// TwinCAT 3 PLC project MTCS
// ProgramVersion: 3.1.4020.1
// libraries:
//   Tc2_ControllerToolbox, * (Beckhoff Automation GmbH)
//   Tc2_Drive, * (Beckhoff Automation GmbH)
//   Tc2_EtherCAT, * (Beckhoff Automation GmbH)
//   Tc2_Math, * (Beckhoff Automation GmbH)
//   Tc2_MC2, * (Beckhoff Automation GmbH)
//   Tc2_MC2_Drive, * (Beckhoff Automation GmbH)
//   Tc2_SerialCom, * (Beckhoff Automation GmbH)
//   Tc2_Standard, * (Beckhoff Automation GmbH)
//   Tc2_System, * (Beckhoff Automation GmbH)
//   Tc2_Utilities, * (Beckhoff Automation GmbH)
//   Tc2_XmlDataSrv, * (Beckhoff Automation GmbH)
//   Tc3_Interfaces, * (Beckhoff Automation GmbH)
//   Tc3_Module, * (Beckhoff Automation GmbH)
//   VisuDialogs, * (System)
//   VisuUserMgmt, * (System)
// project tree:
//   / GlobalTextList.TcGTLO, PlcFastTask.TcTTO, PlcTask.TcTTO, Visualization Manager.TcVMO (not stored), VISU_TASK.TcTTO
//   GVLs/ GLOBAL.TcGVL, REMANENT.TcGVL
//   MTCS/Axes/Generated/mtcs_axes/Configs/ AxesAzimuthConfig.TcDUT (not stored), AxesConfig.TcDUT (not stored), AxesElevationConfig.TcDUT (not stored), AxesKnownPositionConfig.TcDUT (not stored), AxesKnownPositionsConfig.TcDUT (not stored), AxesLocalConditionsConfig.TcDUT (not stored), AxesLocationConfig.TcDUT (not stored), AxesPointingModelConfig.TcDUT (not stored), AxesRotationConfig.TcDUT (not stored)
//   MTCS/Axes/Generated/mtcs_axes/Enums/ AxesAlphaUnits.TcDUT (not stored), AxesDeltaUnits.TcDUT (not stored), AxesIds.TcDUT (not stored), AxesMoveUnits.TcDUT (not stored), AxesMoveVelocityUnits.TcDUT (not stored), AxesMuUnits.TcDUT (not stored), AxesRotatorActivity.TcDUT (not stored)
//   MTCS/Axes/Generated/mtcs_axes/Processes/Args/ AxesEnablePointingModelProcessArgs.TcDUT (not stored), AxesMoveAbsoluteProcessArgs.TcDUT (not stored), AxesMoveKnownPositionProcessArgs.TcDUT (not stored), AxesMoveOutOfLimitSwitchProcessArgs.TcDUT (not stored), AxesMoveRelativeProcessArgs.TcDUT (not stored), AxesMoveVelocityProcessArgs.TcDUT (not stored), AxesMultiMoveProcessArgs.TcDUT (not stored), AxesPointProcessArgs.TcDUT (not stored), AxesPointRelativeProcessArgs.TcDUT (not stored), AxesMultiPowerOnProcessArgs.TcDUT (not stored), AxesSetAlphaDeltaVelocityProcessArgs.TcDUT (not stored), AxesSetPositionProcessArgs.TcDUT (not stored), AxesSetTargetProcessArgs.TcDUT (not stored), AxesUnlockBrakeProcessArgs.TcDUT (not stored)
//   MTCS/Axes/Generated/mtcs_axes/Processes/ AxesDoHomingProcess.TcPOU (not stored), AxesEnablePointingModelProcess.TcPOU (not stored), AxesMoveAbsoluteProcess.TcPOU (not stored), AxesMoveKnownPositionProcess.TcPOU (not stored), AxesMoveOutOfLimitSwitchProcess.TcPOU (not stored), AxesMoveRelativeProcess.TcPOU (not stored), AxesMoveVelocityProcess.TcPOU (not stored), AxesMultiMoveProcess.TcPOU (not stored), AxesPointProcess.TcPOU (not stored), AxesPointRelativeProcess.TcPOU (not stored), AxesPowerOffProcess.TcPOU (not stored), AxesPowerOnProcess.TcPOU (not stored), AxesMultiPowerOnProcess.TcPOU (not stored), AxesSetAlphaDeltaVelocityProcess.TcPOU (not stored), AxesSetPositionProcess.TcPOU (not stored), AxesSetTargetProcess.TcPOU (not stored), AxesStopProcess.TcPOU (not stored), AxesUnlockBrakeProcess.TcPOU (not stored)
//   MTCS/Axes/Generated/mtcs_axes/StateMachines/Parts/ AxesAzimuthAxisParts.TcDUT (not stored), AxesElevationAxisParts.TcDUT (not stored), AxesIOParts.TcDUT (not stored), AxesParts.TcDUT (not stored), AxesPointingModelSetupParts.TcDUT (not stored), AxesPointingModelsSetupParts.TcDUT (not stored), AxesRotationAxisParts.TcDUT (not stored)
//   MTCS/Axes/Generated/mtcs_axes/StateMachines/Processes/ AxesAzimuthAxisProcesses.TcDUT (not stored), AxesElevationAxisProcesses.TcDUT (not stored), AxesProcesses.TcDUT (not stored), AxesRotationAxisProcesses.TcDUT (not stored)
//   MTCS/Axes/Generated/mtcs_axes/StateMachines/ SM_Axes.TcPOU (not stored), SM_AxesAzimuthAxis.TcPOU (not stored), SM_AxesElevationAxis.TcPOU (not stored), SM_AxesFeedback.TcPOU (not stored), SM_AxesIO.TcPOU (not stored), SM_AxesPointingModelSetup.TcPOU (not stored), SM_AxesPointingModelsSetup.TcPOU (not stored), SM_AxesRotationAxis.TcPOU (not stored), SM_AxesTarget.TcPOU (not stored)
//   MTCS/Axes/Generated/mtcs_axes/StateMachines/Statuses/ AxesAzimuthAxisStatuses.TcDUT (not stored), AxesElevationAxisStatuses.TcDUT (not stored), AxesFeedbackStatuses.TcDUT (not stored), AxesIOStatuses.TcDUT (not stored), AxesPointingModelsSetupStatuses.TcDUT (not stored), AxesRotationAxisStatuses.TcDUT (not stored), AxesStatuses.TcDUT (not stored), AxesTargetStatuses.TcDUT (not stored)
//   MTCS/Axes/Helper/ ARCSEC_TO_RAD.TcPOU, AxesDeltaUnitsToDeg.TcPOU, AxesGetKnownPositionConfig.TcPOU, AxesLidaPositionToValue.TcPOU, AxesMoveRelativeCalculator.TcPOU, AxesMoveVelocityUnitsToString.TcPOU, AxesMoveAbsoluteCalculator.TcPOU, AxesSlalibSmoothener.TcPOU, AxesQuickStopHelper.TcPOU, AxesUnlockBrakeHelper.TcPOU, HOUR_TO_DEG.TcPOU, AxesAlphaUnitsToDeg.TcPOU, AxesMoveVelocityUnitsToDegPerSec.TcPOU, HMS_TO_DEG.TcPOU, DEG_TO_ARCSEC.TcPOU, DMS_TO_DEG.TcPOU, MILLIARCSEC_TO_DEG.TcPOU, ARCSEC_TO_DEG.TcPOU, AverageAndRmsCalculator.TcPOU, AxesCalculateLidaAveragePosition.TcPOU, AxesLidaValueToPosition.TcPOU, AxesMuUnitsToDegPerYear.TcPOU, AxesSSIValueToPosition.TcPOU, AxesExternalSetpointGenerator.TcPOU, AxesFastTaskAxisIO.TcDUT, AxesMoveOutOfLimitSwitchHelper.TcPOU, AxesPowerOffHelper.TcPOU, AxesHomingHelper.TcPOU, AxesPowerOnHelper.TcPOU, AxesStopHelper.TcPOU, AxesSetPositionHelper.TcPOU, AxesTorqueSetpointGenerator.TcPOU, AxesCalculateTorqueCommandValue.TcPOU, AxesTPointCalculations.TcPOU, HoursMinutesSeconds.TcDUT, DegreesMinutesSeconds.TcDUT, AxesMoveUnitsToDeg.TcPOU, RAD_TO_DEG.TcPOU, DEG_TO_RAD_REAL.TcPOU, CELSIUS_TO_KELVIN.TcPOU, DEG_TO_RAD.TcPOU, RAD_TO_HOUR.TcPOU, TmcAxesErrorsToString.TcPOU
//   MTCS/Axes/StateMachines/ Axes.TcPOU, AxesElevationAxis.TcPOU, AxesRotationAxis.TcPOU, AxesIO.TcPOU, AxesPointingModelsSetup.TcPOU, AxesAzimuthAxis.TcPOU, AxesPointingModelSetup.TcPOU, AxesTarget.TcPOU, AxesFeedback.TcPOU
//   MTCS/Axes/Visu/Tube/ VISU_Tube_Rotator.TcVIS (not stored), VISU_Tube_Side.TcVIS (not stored), VISU_Tube_Top_0.TcVIS (not stored), VISU_Tube_Top_fork.TcVIS (not stored), VISU_Tube_Top_1.TcVIS (not stored), VISU_Tube_Top_9.TcVIS (not stored), VISU_Tube_Top_10.TcVIS (not stored), VISU_Tube_Top_11.TcVIS (not stored), VISU_Tube_Top_12.TcVIS (not stored), VISU_Tube_Top_14.TcVIS (not stored), VISU_Tube_Top_2.TcVIS (not stored), VISU_Tube_Top_3.TcVIS (not stored), VISU_Tube_Top_13.TcVIS (not stored), VISU_Tube_Top_4.TcVIS (not stored), VISU_Tube_Top_5.TcVIS (not stored), VISU_Tube_Top_6.TcVIS (not stored), VISU_Tube_Top_7.TcVIS (not stored), VISU_Tube_Top_8.TcVIS (not stored), VISU_Tube_Top.TcVIS (not stored)
//   MTCS/Axes/Visu/ VISU_AxesAzimuthAxis.TcVIS, VISU_AxesAzimuthAxis_AbsoluteEncoder.TcVIS, VISU_AxesAzimuthAxis_Processes.TcVIS, VISU_AxesConfig_KnownPosition.TcVIS, VISU_AxesConfig_KnownPositions.TcVIS, VISU_AxesImage.TcVIS, VISU_AxesManual_Offsets_AlphaDeltaRot.TcVIS, VISU_AxesManual_Offsets_OLD.TcVIS, VISU_AxesRotationAxis_Processes.TcVIS, VISU_AxesRotationAxis_Overview.TcVIS, VISU_AxesElevationAxis_Processes.TcVIS, VISU_AxesManual_MoveVelocity.TcVIS, VISU_AxesManual_Offsets_AziEleRot.TcVIS, VISU_AxesManual_Joystick_AziEle.TcVIS, VISU_AxesManual_Joystick_Rot.TcVIS, VISU_AxesManual_Positions.TcVIS, VISU_AxesManual_MoveAbsolute.TcVIS, VISU_Axes_Commands_Power.TcVIS, VISU_AxesElevationAxis_Overview.TcVIS, VISU_AxesElevationAxis_AbsoluteEncoder.TcVIS, VISU_AxesElevationAxis_Lidas.TcVIS, VISU_AxesAzimuthAxis_Overview.TcVIS, VISU_AxesAzimuthAxis_Lidas.TcVIS, VISU_AxesConfig_Azimuth_1.TcVIS, VISU_AxesConfig_Azimuth_3.TcVIS, VISU_AxesConfig_Rotation_2.TcVIS, VISU_AxesConfig_Rotation_1.TcVIS, VISU_AxesConfig_Elevation_2.TcVIS, VISU_AxesConfig_Elevation_1.TcVIS, VISU_AxesConfig_Azimuth_2.TcVIS, VISU_AxesConfig_FilterWheel.TcVIS, VISU_AxesElevationAxis.TcVIS, VISU_AxesExternalSetpointGenerator.TcVIS, VISU_AxesRotationAxis.TcVIS, VISU_AxesManual.TcVIS, VISU_AxesConfig.TcVIS, VISU_AxesAxes.TcVIS, VISU_AxesAdvanced.TcVIS, VISU_AxesPointingModelConfig_part1.TcVIS, VISU_AxesPointingModelConfig_part2.TcVIS, VISU_AxesPointingModelSetup.TcVIS, VISU_AxesConfig_General.TcVIS, VISU_AxesConfig_Location.TcVIS, VISU_AxesConfig_LocalConditions.TcVIS, VISU_AxesFromCpp_Target.TcVIS, VISU_AxesIO.TcVIS, VISU_Axes.TcVIS, VISU_AxesOverview.TcVIS, VISU_AxesMultiMoveProcess.TcVIS, VISU_AxesPointingModelsSetup.TcVIS, VISU_AxesPointDialog.TcVIS, VISU_AxesTarget.TcVIS, VISU_AxesSetTargetDialog.TcVIS, VISU_AxesFromCpp.TcVIS, VISU_Axes_Commands_Reset.TcVIS, VISU_Axes_Commands_Brake.TcVIS, VISU_Axes_Commands_Movement.TcVIS, VISU_Axes_Commands_DoHoming.TcVIS, VISU_Axes_stats.TcVIS
//   MTCS/Axes/Widgets/ AxesAlphaWidget.TcPOU, AxesAngleWidget.TcPOU, AxesDialogRotUnits.TcDUT, AxesDialogRotUnitsTextList.TcTLO, AxesMoveAlphaDeltaProcessUnitsTextList.TcTLO, AxesPointRelativeProcessWidget.TcPOU, AxesRotationAxisTabs.TcDUT, AxesManualTabs.TcDUT, AxesElevationAxisTabs.TcDUT, AxesDeltaWidget.TcPOU, AxesAzimuthAxisTabs.TcDUT, AxesDialogAlphaUnitsTextList.TcTLO, AxesDialogSignTextList.TcTLO, AxesManualJoystickAziEleWidget.TcPOU, AxesManualJoystickRotWidget.TcPOU, AxesManualOffsetsWidget.TcPOU, AxesManualMoveVelocityWidget.TcPOU, AxesManualPositionsWidget.TcPOU, AxesManualMoveAbsoluteWidget.TcPOU, AxesMoveUnitsTextList.TcTLO, AxesMoveVelocityUnitsTextList.TcTLO, AxesMuUnitsTextList.TcTLO, AxesDialogDeltaUnitsTextList.TcTLO, AxesDialogSign.TcDUT, AxesElevationAxisWidget.TcPOU, AxesConfigTextList.TcTLO, AxesAxesTabs.TcDUT, AxesAxesWidget.TcPOU, AxesImageWidget.TcPOU, AxesManualWidget.TcPOU, AxesMultiMoveProcessWidget.TcPOU, AxesRotationAxisWidget.TcPOU, AxesPointingModelSetupPartsTextList.TcTLO, AxesIOWidget.TcPOU, AxesPointingModelSetupWidget.TcPOU, AxesMoveProcessUnitsTextList.TcTLO, AxesMoveProcessWidgetUnits.TcDUT, AxesPointingModelsSetupWidget.TcPOU, AxesAzimuthAxisWidget.TcPOU, AxesDialogAlphaUnits.TcDUT, AxesDialogDeltaUnits.TcDUT, AxesSetTargetDialogWidget.TcPOU, AxesPointDialogWidget.TcPOU, AxesTabs.TcDUT, AxesTargetWidget.TcPOU, AxesFeedbackWidget.TcPOU, AxesWidget.TcPOU
//   MTCS/Common/Generated/mtcs_common/Configs/ FaulhaberDriveConfig.TcDUT (not stored), HiHiLoLoAlarmConfig.TcDUT (not stored), InstrumentConfig.TcDUT (not stored), MeasurementConfig.TcDUT (not stored)
//   MTCS/Common/Generated/mtcs_common/Enums/ DriveBrakeStates.TcDUT (not stored), DriveOperatingModes.TcDUT (not stored), InitializationStates.TcDUT (not stored), LimitSwitches.TcDUT (not stored), OperatingStates.TcDUT (not stored), OperatorStates.TcDUT (not stored), RequestResults.TcDUT (not stored), Units.TcDUT (not stored)
//   MTCS/Common/Generated/mtcs_common/Processes/ ActivateProcess.TcPOU (not stored), ChangeOperatingStateProcess.TcPOU (not stored), ChangeOperatorStateProcess.TcPOU (not stored), ChangeSetpointProcess.TcPOU (not stored), McMoveAbsoluteProcess.TcPOU (not stored), McMoveRelativeProcess.TcPOU (not stored), McMoveVelocityProcess.TcPOU (not stored), McPowerProcess.TcPOU (not stored), McProcess.TcPOU (not stored), McReadBoolParameter.TcPOU (not stored), McReadParameter.TcPOU (not stored), McSetPositionProcess.TcPOU (not stored), McStopProcess.TcPOU (not stored), McWriteBoolParameter.TcPOU (not stored), McWriteParameter.TcPOU (not stored), Process.TcPOU (not stored), ReadXmlProcess.TcPOU (not stored), SDOReadProcess.TcPOU (not stored), SDOWriteProcess.TcPOU (not stored), SetBrakeProcess.TcPOU (not stored), SetEnabledProcess.TcPOU (not stored), SoEReadProcess.TcPOU (not stored), SoEResetProcess.TcPOU (not stored), SoEWriteProcess.TcPOU (not stored), WriteXmlProcess.TcPOU (not stored)
//   MTCS/Common/Generated/mtcs_common/Processes/Args/ ChangeOperatingStateProcessArgs.TcDUT (not stored), ChangeOperatorStateProcessArgs.TcDUT (not stored), ChangeSetpointProcessArgs.TcDUT (not stored), McMoveAbsoluteProcessArgs.TcDUT (not stored), McMoveRelativeProcessArgs.TcDUT (not stored), McMoveVelocityProcessArgs.TcDUT (not stored), McPowerProcessArgs.TcDUT (not stored), McReadBoolParameterArgs.TcDUT (not stored), McReadParameterArgs.TcDUT (not stored), McSetPositionProcessArgs.TcDUT (not stored), McStopProcessArgs.TcDUT (not stored), McWriteBoolParameterArgs.TcDUT (not stored), McWriteParameterArgs.TcDUT (not stored), ReadXmlProcessArgs.TcDUT (not stored), SDOReadProcessArgs.TcDUT (not stored), SDOWriteProcessArgs.TcDUT (not stored), SetBrakeProcessArgs.TcDUT (not stored), SetEnabledProcessArgs.TcDUT (not stored), SoEReadProcessArgs.TcDUT (not stored), SoEWriteProcessArgs.TcDUT (not stored), WriteXmlProcessArgs.TcDUT (not stored)
//   MTCS/Common/Generated/mtcs_common/StateMachines/Parts/ AX52XXDriveParts.TcDUT (not stored)
//   MTCS/Common/Generated/mtcs_common/StateMachines/Processes/ AX52XXDriveChannelProcesses.TcDUT (not stored), BaseAxisProcesses.TcDUT (not stored), ConfigManagerProcesses.TcDUT (not stored), FaulhaberDriveProcesses.TcDUT (not stored), IncrementalEncoderProcesses.TcDUT (not stored), SimpleRelayProcesses.TcDUT (not stored)
//   MTCS/Common/Generated/mtcs_common/StateMachines/ SM_AngularAcceleration.TcPOU (not stored), SM_AngularAxis.TcPOU (not stored), SM_AngularPosition.TcPOU (not stored), SM_AngularVelocity.TcPOU (not stored), SM_AverageCurrent.TcPOU (not stored), SM_AX52XXDrive.TcPOU (not stored), SM_AX52XXDriveChannel.TcPOU (not stored), SM_BaseAxis.TcPOU (not stored), SM_BaseMcProcess.TcPOU (not stored), SM_BaseProcess.TcPOU (not stored), SM_BaseXmlDataSrvProcess.TcPOU (not stored), SM_CANopenBus.TcPOU (not stored), SM_ConfigManager.TcPOU (not stored), SM_Current.TcPOU (not stored), SM_CurrentMeasurement.TcPOU (not stored), SM_EtherCatDevice.TcPOU (not stored), SM_FaulhaberDrive.TcPOU (not stored), SM_Force.TcPOU (not stored), SM_ForceMeasurement.TcPOU (not stored), SM_Fraction.TcPOU (not stored), SM_Frequency.TcPOU (not stored), SM_FrequencyMeasurement.TcPOU (not stored), SM_GForce.TcPOU (not stored), SM_GForceMeasurement.TcPOU (not stored), SM_IncrementalEncoder.TcPOU (not stored), SM_LinearAxis.TcPOU (not stored), SM_LinearPosition.TcPOU (not stored), SM_LinearPositionMeasurement16.TcPOU (not stored), SM_LinearPositionMeasurementU32.TcPOU (not stored), SM_LinearVelocity.TcPOU (not stored), SM_Pressure.TcPOU (not stored), SM_PressureMeasurement.TcPOU (not stored), SM_ProcessStep.TcPOU (not stored), SM_QuantityValue.TcPOU (not stored), SM_RelativeHumidityMeasurement.TcPOU (not stored), SM_SimpleRelay.TcPOU (not stored), SM_SSIEncoder.TcPOU (not stored), SM_Temperature.TcPOU (not stored), SM_TemperatureMeasurement.TcPOU (not stored), SM_Torque.TcPOU (not stored), SM_TorqueLimit.TcPOU (not stored), SM_Voltage.TcPOU (not stored), SM_VoltageMeasurement.TcPOU (not stored)
//   MTCS/Common/Generated/mtcs_common/StateMachines/Statuses/ AX52XXDriveChannelStatuses.TcDUT (not stored), AX52XXDriveStatuses.TcDUT (not stored), BaseAxisStatuses.TcDUT (not stored), BaseProcessStatuses.TcDUT (not stored), CANopenBusStatuses.TcDUT (not stored), ConfigManagerStatuses.TcDUT (not stored), CurrentMeasurementStatuses.TcDUT (not stored), EtherCatDeviceStatuses.TcDUT (not stored), FaulhaberDriveStatuses.TcDUT (not stored), ForceMeasurementStatuses.TcDUT (not stored), FrequencyMeasurementStatuses.TcDUT (not stored), GForceMeasurementStatuses.TcDUT (not stored), IncrementalEncoderStatuses.TcDUT (not stored), LinearPositionMeasurement16Statuses.TcDUT (not stored), LinearPositionMeasurementU32Statuses.TcDUT (not stored), PressureMeasurementStatuses.TcDUT (not stored), ProcessStepStatuses.TcDUT (not stored), RelativeHumidityMeasurementStatuses.TcDUT (not stored), SimpleRelayStatuses.TcDUT (not stored), SSIEncoderStatuses.TcDUT (not stored), TemperatureMeasurementStatuses.TcDUT (not stored), VoltageMeasurementStatuses.TcDUT (not stored)
//   MTCS/Common/Generated/mtcs_common/Statuses/ ActivityStatus.TcPOU (not stored), ApertureStatus.TcPOU (not stored), BusyStatus.TcPOU (not stored), EnabledStatus.TcPOU (not stored), HealthStatus.TcPOU (not stored), HiHiLoLoAlarmStatus.TcPOU (not stored), InitializationStatus.TcPOU (not stored), MotionStatus.TcPOU (not stored), OpeningStatus.TcPOU (not stored), OperatingStatus.TcPOU (not stored), OperatorStatus.TcPOU (not stored), PoweredStatus.TcPOU (not stored), StartedStatus.TcPOU (not stored)
//   MTCS/Common/HelperCode/ BusyToColor.TcPOU, ComErrorToString.TcPOU, DegToRad.TcPOU, DriveBrakeStatesToString.TcPOU, DriveOperatingModesToString.TcPOU, HealthBusyToColor.TcPOU, HealthToColor.TcPOU, InitializationStatusToString.TcPOU, MeasurementToString.TcPOU, MeasurementToStatus.TcPOU, RadToDeg.TcPOU, SerialLine.TcPOU, StatusColor.TcDUT, SystemToColor.TcPOU
//   MTCS/Common/StateMachines/ AngularAxis.TcPOU, AngularPosition.TcPOU, AngularVelocity.TcPOU, AngularAcceleration.TcPOU, AverageCurrent.TcPOU, AX52XXDrive.TcPOU, AX52XXDriveChannel.TcPOU, BaseAxis.TcPOU, BaseMcProcess.TcPOU, BaseProcess.TcPOU, BaseXmlDataSrvProcess.TcPOU, CANopenBus.TcPOU, ConfigManager.TcPOU, Current.TcPOU, CurrentMeasurement.TcPOU, Torque.TcPOU, GForce.TcPOU, LinearPositionMeasurement16.TcPOU, EtherCatDevice.TcPOU, FaulhaberDrive.TcPOU, Force.TcPOU, ForceMeasurement.TcPOU, Frequency.TcPOU, FrequencyMeasurement.TcPOU, Fraction.TcPOU, IncrementalEncoder.TcPOU, LinearAxis.TcPOU, LinearPosition.TcPOU, LinearPositionMeasurementU32.TcPOU, LinearVelocity.TcPOU, Pressure.TcPOU, PressureMeasurement.TcPOU, ProcessStep.TcPOU, QuantityValue.TcPOU, RelativeHumidityMeasurement.TcPOU, SimpleRelay.TcPOU, SSIEncoder.TcPOU, Temperature.TcPOU, TemperatureMeasurement.TcPOU, TorqueLimit.TcPOU, Voltage.TcPOU, VoltageMeasurement.TcPOU, GForceMeasurement.TcPOU
//   MTCS/Common/Visu/ VISU_AX522Drive.TcVIS, VISU_BaseAxis_Gearing.TcVIS, VISU_BaseAxis_MoveVelocity.TcVIS, VISU_ConfigBOOLEntry_Small.TcVIS, VISU_ConfigDINTEntry.TcVIS, VISU_ConfigREAL4Entry.TcVIS, VISU_ConfigLREAL8Entry.TcVIS, VISU_ConfigLREAL1Entry.TcVIS, VISU_ConfigUINTEntry.TcVIS, VISU_ConfigBOOLEntry.TcVIS, VISU_ConfigLREAL4Entry.TcVIS, VISU_ConfigUDINTEntry.TcVIS, VISU_ConfigINTEntry.TcVIS, VISU_ConfigUSINTEntry.TcVIS, VISU_CANopenBus.TcVIS, VISU_ConfigSINTEntry.TcVIS, VISU_EtherCatFillerDevice.TcVIS, VISU_AX522DriveChannel.TcVIS, VISU_FaulhaberDriveConfig.TcVIS, VISU_FaulhaberDrive.TcVIS, VISU_ConfigStringEntry.TcVIS, VISU_FaulhaberDriveConfig_LimitSwitches.TcVIS, VISU_FaulhaberDriveConfig_General.TcVIS, VISU_FaulhaberDriveConfig_Control.TcVIS, VISU_FaulhaberDrive_SDOWrite.TcVIS, VISU_HiHiLoLoAlarmConfig.TcVIS, VISU_IncrementalEncoder.TcVIS, VISU_IvsLogo.TcIPO (not stored), VISU_LinearAxis.TcVIS, VISU_BaseAxis_Stop.TcVIS, VISU_FaulhaberDrive_SDORead.TcVIS, VISU_BaseAxis_MoveAbsolute.TcVIS, VISU_BaseAxis_Power.TcVIS, VISU_BaseAxis_Status.TcVIS, VISU_ConfigManager.TcVIS, VISU_EtherCatDevice.TcVIS, VISU_Measurement.TcVIS, VISU_MeasurementConfig.TcVIS, VISU_ProcessStep.TcVIS, VISU_SimpleRelay.TcVIS, VISU_SSIEncoder.TcVIS, VISU_State_gray_yellow.TcVIS, VISU_State_gray_red.TcVIS, VISU_State_green_gray.TcVIS, VISU_StatusWidget.TcVIS, VISU_AngularAxis.TcVIS, VISU_OperatingStatus.TcVIS, VISU_OperatorStatus.TcVIS, VISU_OperatorStatus_Old.TcVIS, VISU_State.TcVIS, VISU_State_gray_green.TcVIS, VISU_State_gray_orange.TcVIS, VISU_State_green_red.TcVIS, VISU_State_red_green.TcVIS, VISU_SubSubSystemButton.TcVIS, VISU_SystemBackground.TcVIS, VISU_SystemButton.TcVIS, VISU_SubSystemButton.TcVIS, VISU_SystemButtonImages.TcIPO (not stored), VISU_SystemButton_backup.TcVIS, VISU_SystemControl.TcVIS
//   MTCS/Common/Widgets/ AngularAxisWidget.TcPOU, AX52XXDriveWidget.TcPOU, AX52XXDriveChannelWidget.TcPOU, BaseAxisWidget.TcPOU, CANopenBusWidget.TcPOU, Colors.TcDUT, ConfigManagerWidget.TcPOU, EtherCatDeviceWidget.TcPOU, FaulhaberDriveWidget.TcPOU, IncrementalEncoderWidget.TcPOU, InitializationStatusWidget.TcPOU, ActivityStatusWidget.TcPOU, InitializeButtonWidget.TcPOU, LimitSwitchesTextList.TcTLO, LinearAxisWidget.TcPOU, LockingButtonWidget.TcPOU, ActivityButtonWidget.TcPOU, McProcessWidget.TcPOU, MeasurementWidget.TcPOU, OperatingButtonWidget.TcPOU, ProcessStepWidget.TcPOU, ReadXmlProcessWidget.TcPOU, SimpleRelayWidget.TcPOU, StatusWidget.TcPOU, SubSubSystemButtonWidget.TcPOU, SubSystemButtonWidget.TcPOU, SystemButtonWidget.TcPOU, WriteXmlProcessWidget.TcPOU
//   MTCS/Cover/Generated/mtcs_cover/Configs/ CoverConfig.TcDUT (not stored), CoverPanelConfig.TcDUT (not stored), CoverPanelSetConfig.TcDUT (not stored)
//   MTCS/Cover/Generated/mtcs_cover/Enums/ CoverApertureProcedureStates.TcDUT (not stored)
//   MTCS/Cover/Generated/mtcs_cover/StateMachines/Parts/ CoverIOParts.TcDUT (not stored), CoverPanelParts.TcDUT (not stored), CoverPanelSetParts.TcDUT (not stored), CoverParts.TcDUT (not stored)
//   MTCS/Cover/Generated/mtcs_cover/StateMachines/Processes/ CoverPanelProcesses.TcDUT (not stored), CoverPanelSetProcesses.TcDUT (not stored), CoverProcesses.TcDUT (not stored)
//   MTCS/Cover/Generated/mtcs_cover/StateMachines/ SM_Cover.TcPOU (not stored), SM_CoverApertureProcedure.TcPOU (not stored), SM_CoverIO.TcPOU (not stored), SM_CoverPanel.TcPOU (not stored), SM_CoverPanelSet.TcPOU (not stored)
//   MTCS/Cover/Generated/mtcs_cover/StateMachines/Statuses/ CoverApertureProcedureStatuses.TcDUT (not stored), CoverIOStatuses.TcDUT (not stored), CoverPanelSetStatuses.TcDUT (not stored), CoverPanelStatuses.TcDUT (not stored), CoverStatuses.TcDUT (not stored)
//   MTCS/Cover/StateMachines/ Cover.TcPOU, CoverApertureProcedure.TcPOU, CoverIO.TcPOU, CoverPanel.TcPOU, CoverPanelSet.TcPOU
//   MTCS/Cover/Visu/ VISU_Cover.TcVIS, VISU_CoverConfig_General.TcVIS, VISU_CoverConfig_Panel.TcVIS (not stored), VISU_CoverPanelOverviewDrawing.TcVIS (not stored), VISU_CoverConfig.TcVIS, VISU_CoverIO.TcVIS (not stored), VISU_CoverIOSmall.TcVIS (not stored), VISU_CoverPanel.TcVIS (not stored), VISU_CoverPanelConfig.TcVIS (not stored), VISU_CoverPanelDetails.TcVIS (not stored), VISU_CoverPanelDrawing.TcVIS (not stored), VISU_CoverPanelSet.TcVIS (not stored), VISU_CoverConfig_PanelSet.TcVIS, VISU_COVER_OVERVIEW.TcVIS
//   MTCS/Cover/Widgets/ CoverConfigTabs.TcDUT, CoverConfigTabsTextList.TcTLO, CoverIOWidget.TcPOU, CoverPanelSetWidget.TcPOU, CoverPanelWidget.TcPOU, CoverTabs.TcDUT, CoverWidget.TcPOU
//   MTCS/Hydraulics/Generated/mtcs_hydraulics/Configs/ HydraulicsConfig.TcDUT (not stored), HydraulicsSideConfig.TcDUT (not stored)
//   MTCS/Hydraulics/Generated/mtcs_hydraulics/Enums/ HydraulicsPumpsStates.TcDUT (not stored)
//   MTCS/Hydraulics/Generated/mtcs_hydraulics/StateMachines/Parts/ HydraulicsIOParts.TcDUT (not stored), HydraulicsParts.TcDUT (not stored), HydraulicsPumpsGroupIOParts.TcDUT (not stored)
//   MTCS/Hydraulics/Generated/mtcs_hydraulics/StateMachines/Processes/ HydraulicsProcesses.TcDUT (not stored), HydraulicsSideProcesses.TcDUT (not stored)
//   MTCS/Hydraulics/Generated/mtcs_hydraulics/StateMachines/ SM_Hydraulics.TcPOU (not stored), SM_HydraulicsIO.TcPOU (not stored), SM_HydraulicsPumpsGroupIO.TcPOU (not stored), SM_HydraulicsSide.TcPOU (not stored)
//   MTCS/Hydraulics/Generated/mtcs_hydraulics/StateMachines/Statuses/ HydraulicsIOStatuses.TcDUT (not stored), HydraulicsPumpsGroupIOStatuses.TcDUT (not stored), HydraulicsSideStatuses.TcDUT (not stored), HydraulicsStatuses.TcDUT (not stored)
//   MTCS/Hydraulics/StateMachines/ Hydraulics.TcPOU, HydraulicsIO.TcPOU, HydraulicsPumpsGroupIO.TcPOU, HydraulicsSide.TcPOU
//   MTCS/Hydraulics/Visu/ VISU_HydraulicsPumpsGroupIO.TcVIS (not stored), VISU_HydraulicsMeasurements.TcVIS (not stored), VISU_HydraulicsConfig_General.TcVIS (not stored), VISU_HydraulicsConfig_Side_General.TcVIS (not stored), VISU_HydraulicsFigure.TcVIS (not stored), VISU_HydraulicsFigure_Manometer.TcVIS (not stored), VISU_HydraulicsFigure_Pipe.TcVIS (not stored), VISU_Hydraulics.TcVIS (not stored), VISU_HydraulicsSafety.TcVIS (not stored), VISU_HydraulicsPumpsStatus.TcVIS (not stored), VISU_HydraulicsTechnical.TcVIS (not stored), VISU_HydraulicsOverview.TcVIS (not stored), VISU_HydraulicsIO.TcVIS (not stored), VISU_HydraulicsConfig.TcVIS (not stored), VISU_HydraulicsChangeFrequencies.TcVIS (not stored)
//   MTCS/Hydraulics/Widgets/ HydraulicsSideWidget.TcPOU, HydraulicsTabs.TcDUT, HydraulicsIOWidget.TcPOU, HydraulicsWidget.TcPOU, HydraulicsConfigTabsTextList.TcTLO, HydraulicsPumpsGroupIOWidget.TcPOU
//   MTCS/M1/Generated/mtcs_m1/Configs/ M1AxialSupportConfig.TcDUT (not stored), M1Config.TcDUT (not stored), M1RadialSupportConfig.TcDUT (not stored)
//   MTCS/M1/Generated/mtcs_m1/StateMachines/Parts/ M1M2IOParts.TcDUT (not stored), M1Parts.TcDUT (not stored), M1RadialSupportParts.TcDUT (not stored)
//   MTCS/M1/Generated/mtcs_m1/StateMachines/Processes/ M1AxialSupportProcesses.TcDUT (not stored), M1Processes.TcDUT (not stored), M1RadialSupportProcesses.TcDUT (not stored)
//   MTCS/M1/Generated/mtcs_m1/StateMachines/ SM_M1.TcPOU (not stored), SM_M1AxialSupport.TcPOU (not stored), SM_M1Inclinometer.TcPOU (not stored), SM_M1M2IO.TcPOU (not stored), SM_M1RadialSupport.TcPOU (not stored)
//   MTCS/M1/Generated/mtcs_m1/StateMachines/Statuses/ M1AxialSupportStatuses.TcDUT (not stored), M1InclinometerStatuses.TcDUT (not stored), M1M2IOStatuses.TcDUT (not stored), M1RadialSupportStatuses.TcDUT (not stored), M1Statuses.TcDUT (not stored)
//   MTCS/M1/StateMachines/ M1.TcPOU, M1AxialSupport.TcPOU, M1Inclinometer.TcPOU, M1M2IO.TcPOU, M1RadialSupport.TcPOU
//   MTCS/M1/Visu/ VISU_M1.TcVIS (not stored), VISU_M1AxialSupportController.TcVIS (not stored), VISU_M1Config_Axial_ForceSensors.TcVIS (not stored), VISU_M1Config_Axial_AverageForce.TcVIS (not stored), VISU_M1Config_General.TcVIS (not stored), VISU_M1Config_Axial_General.TcVIS (not stored), VISU_M1Config_Axial_MirrorPressure.TcVIS (not stored), VISU_M1Config_Radial_RegulatorPressure.TcVIS (not stored), VISU_M1Config_Radial_MirrorPressure.TcVIS (not stored), VISU_M1Config_Radial_General.TcVIS (not stored), VISU_M1Config_Axial_RegulatorPressure.TcVIS (not stored), VISU_M1Figure_Dryer.TcVIS (not stored), VISU_M1Figure_Gauge.TcVIS (not stored), VISU_M1Figure_Supply.TcVIS (not stored), VISU_M1Figure_Valve.TcVIS (not stored), VISU_M1Figure_Regulator.TcVIS (not stored), VISU_M1Figure_FilterWithDrain.TcVIS (not stored), VISU_M1M2IO.TcVIS (not stored), VISU_M1Overview.TcVIS (not stored), VISU_M1Figure.TcVIS (not stored), VISU_M1FullFigure.TcVIS (not stored), VISU_M1RadialSupport.TcVIS (not stored), VISU_M1AxialSupport.TcVIS (not stored), VISU_M1Config.TcVIS (not stored), VISU_M1AxialSupportSetpoint.TcVIS (not stored), VISU_M1RadialSupportVacuum.TcVIS (not stored), VISU_M1RadialSupportStatus.TcVIS (not stored), VISU_M1RadialSupportSetpoint.TcVIS (not stored)
//   MTCS/M1/Widgets/ M1AxialSupportWidget.TcPOU, M1ConfigTabsTextList.TcTLO, M1FigureWidget.TcPOU, M1RadialSupportWidget.TcPOU, M1M2IOWidget.TcPOU, M1InclinometerWidget.TcPOU, M1Widget.TcPOU, M1Tabs.TcDUT
//   MTCS/M2/Generated/mtcs_m2/Configs/ M2AxisGeneralConfig.TcDUT (not stored), M2Config.TcDUT (not stored), M2ConstantsTiltX.TcDUT (not stored), M2ConstantsTiltY.TcDUT (not stored), M2ConstantsX.TcDUT (not stored), M2ConstantsY.TcDUT (not stored), M2ConstantsZ.TcDUT (not stored), M2PotentiometerAxisConfig.TcDUT (not stored), M2ThermalFocusConfig.TcDUT (not stored), M2ThermalFocusStationConfig.TcDUT (not stored), M2ZAxisConfig.TcDUT (not stored)
//   MTCS/M2/Generated/mtcs_m2/Enums/ M2Axes.TcDUT (not stored), M2MoveProcedureStates.TcDUT (not stored)
//   MTCS/M2/Generated/mtcs_m2/Processes/Args/ M2DoThermalFocusForStationNameArgs.TcDUT (not stored), M2DoThermalFocusForStationPositionArgs.TcDUT (not stored), M2MoveProcessArgs.TcDUT (not stored), M2MoveStepsProcessArgs.TcDUT (not stored), M2SelectAxisProcessArgs.TcDUT (not stored)
//   MTCS/M2/Generated/mtcs_m2/Processes/ M2DoThermalFocusForStationName.TcPOU (not stored), M2DoThermalFocusForStationPosition.TcPOU (not stored), M2MoveProcess.TcPOU (not stored), M2MoveStepsProcess.TcPOU (not stored), M2SelectAxisProcess.TcPOU (not stored)
//   MTCS/M2/Generated/mtcs_m2/StateMachines/Parts/ M2MultiplexerParts.TcDUT (not stored), M2Parts.TcDUT (not stored), M2ZAxisParts.TcDUT (not stored)
//   MTCS/M2/Generated/mtcs_m2/StateMachines/Processes/ M2MultiplexerProcesses.TcDUT (not stored), M2Processes.TcDUT (not stored)
//   MTCS/M2/Generated/mtcs_m2/StateMachines/ SM_M2.TcPOU (not stored), SM_M2MovePositionProcedure.TcPOU (not stored), SM_M2MoveStepsProcedure.TcPOU (not stored), SM_M2Multiplexer.TcPOU (not stored), SM_M2TiltXAxis.TcPOU (not stored), SM_M2TiltYAxis.TcPOU (not stored), SM_M2XAxis.TcPOU (not stored), SM_M2YAxis.TcPOU (not stored), SM_M2ZAxis.TcPOU (not stored)
//   MTCS/M2/Generated/mtcs_m2/StateMachines/Statuses/ M2MovePositionProcedureStatuses.TcDUT (not stored), M2MoveStepsProcedureStatuses.TcDUT (not stored), M2MultiplexerStatuses.TcDUT (not stored), M2Statuses.TcDUT (not stored), M2TiltXAxisStatuses.TcDUT (not stored), M2TiltYAxisStatuses.TcDUT (not stored), M2XAxisStatuses.TcDUT (not stored), M2YAxisStatuses.TcDUT (not stored), M2ZAxisStatuses.TcDUT (not stored)
//   MTCS/M2/Helper/ M2AxisToAddress.TcPOU, M2AddressToAxis.TcPOU, M2AxisToGeneralConfig.TcPOU, M2AxisToString.TcPOU, M2ComputeAbsoluteMove.TcPOU, M2ComputeThermalFocusFromId.TcPOU, M2FastTaskControl.TcPOU (not stored), M2ComputeThermalFocus.TcPOU
//   MTCS/M2/StateMachines/ M2.TcPOU (not stored), M2MovePositionProcedure.TcPOU (not stored), M2MoveStepsProcedure.TcPOU (not stored), M2XAxis.TcPOU (not stored), M2Multiplexer.TcPOU (not stored), M2YAxis.TcPOU (not stored), M2ZAxis.TcPOU (not stored), M2TiltXAxis.TcPOU, M2TiltYAxis.TcPOU (not stored)
//   MTCS/M2/Visu/ VISU_M2AxisControl.TcVIS (not stored), VISU_M2Fixed.TcVIS (not stored), VISU_M2ZAxisControl.TcVIS (not stored), VISU_M2Config_General.TcVIS (not stored), VISU_M2Config.TcVIS (not stored), VISU_M2.TcVIS (not stored), VISU_M2Config_PotentiometerAxis.TcVIS (not stored), VISU_M2Config_AxisGeneral.TcVIS (not stored), VISU_M2Config_ZAxis_General.TcVIS (not stored), VISU_M2Config_ThermalFocus.TcVIS (not stored), VISU_M2Config_ThermalFocusStation.TcVIS (not stored), VISU_M2Config_ZAxis_Specific.TcVIS (not stored), VISU_M2Figure.TcVIS (not stored), VISU_M2MoveSteps.TcVIS (not stored), VISU_M2Multiplexer.TcVIS (not stored), VISU_M2Power.TcVIS (not stored), VISU_M2Overview.TcVIS (not stored), VISU_M2Procedures.TcVIS (not stored), VISU_M2ThermalFocus.TcVIS (not stored), VISU_M2Technical.TcVIS (not stored), VISU_M2Axes.TcVIS (not stored)
//   MTCS/M2/Widgets/ M2AxesTextList.TcTLO (not stored), M2AxisWidget.TcPOU (not stored), M2MoveStepsWidget.TcPOU (not stored), M2MovePositionWidget.TcPOU (not stored), M2Tabs.TcDUT (not stored), M2Widget.TcPOU (not stored), M2ConfigTabsTextList.TcTLO (not stored), M2FigureWidget.TcPOU (not stored), M2MultiplexerWidget.TcPOU (not stored)
//   MTCS/M3/Generated/mtcs_m3/Configs/ M3Config.TcDUT (not stored), M3KnownPositionsConfig.TcDUT (not stored), M3PositionConfig.TcDUT (not stored), M3RotationConfig.TcDUT (not stored), M3TranslationConfig.TcDUT (not stored)
//   MTCS/M3/Generated/mtcs_m3/Enums/ M3CalibrateRotationProcedureStates.TcDUT (not stored), M3GotoProcedureStates.TcDUT (not stored), M3PositionIDs.TcDUT (not stored), M3RotateProcedureStates.TcDUT (not stored), M3TargetStates.TcDUT (not stored), M3TranslateProcedureStates.TcDUT (not stored), M3TranslationHomingProcedureStates.TcDUT (not stored)
//   MTCS/M3/Generated/mtcs_m3/Processes/Args/ M3GotoKnownPositionArgs.TcDUT (not stored), M3GotoNewPositionArgs.TcDUT (not stored), M3RotationGotoArgs.TcDUT (not stored), M3TranslationGotoArgs.TcDUT (not stored)
//   MTCS/M3/Generated/mtcs_m3/Processes/ M3GotoKnownPosition.TcPOU (not stored), M3GotoNewPosition.TcPOU (not stored), M3RotationGoto.TcPOU (not stored), M3TranslationGoto.TcPOU (not stored)
//   MTCS/M3/Generated/mtcs_m3/StateMachines/Parts/ M3IOParts.TcDUT (not stored), M3Parts.TcDUT (not stored), M3RotationParts.TcDUT (not stored), M3TranslationParts.TcDUT (not stored)
//   MTCS/M3/Generated/mtcs_m3/StateMachines/Processes/ M3Processes.TcDUT (not stored), M3RotationProcesses.TcDUT (not stored), M3TranslationProcesses.TcDUT (not stored)
//   MTCS/M3/Generated/mtcs_m3/StateMachines/ SM_M3.TcPOU (not stored), SM_M3GotoProcedure.TcPOU (not stored), SM_M3IO.TcPOU (not stored), SM_M3Rotation.TcPOU (not stored), SM_M3RotationCalibrateProcedure.TcPOU (not stored), SM_M3RotationGotoProcedure.TcPOU (not stored), SM_M3RotationTarget.TcPOU (not stored), SM_M3Translation.TcPOU (not stored), SM_M3TranslationGotoProcedure.TcPOU (not stored), SM_M3TranslationHomingProcedure.TcPOU (not stored), SM_M3TranslationTarget.TcPOU (not stored)
//   MTCS/M3/Generated/mtcs_m3/StateMachines/Statuses/ M3GotoProcedureStatuses.TcDUT (not stored), M3IOStatuses.TcDUT (not stored), M3RotationCalibrateProcedureStatuses.TcDUT (not stored), M3RotationGotoProcedureStatuses.TcDUT (not stored), M3RotationStatuses.TcDUT (not stored), M3RotationTargetStatuses.TcDUT (not stored), M3Statuses.TcDUT (not stored), M3TranslationGotoProcedureStatuses.TcDUT (not stored), M3TranslationHomingProcedureStatuses.TcDUT (not stored), M3TranslationStatuses.TcDUT (not stored), M3TranslationTargetStatuses.TcDUT (not stored)
//   MTCS/M3/Generated/mtcs_m3/Statuses/ M3TargetStatus.TcPOU (not stored)
//   MTCS/M3/Helper/ M3PositionIDToName.TcPOU (not stored), M3NameToPositionId.TcPOU (not stored)
//   MTCS/M3/StateMachines/ M3.TcPOU (not stored), M3GotoProcedure.TcPOU (not stored), M3IO.TcPOU (not stored), M3Rotation.TcPOU (not stored), M3RotationCalibrateProcedure.TcPOU (not stored), M3RotationGotoProcedure.TcPOU (not stored), M3RotationTarget.TcPOU (not stored), M3Translation.TcPOU (not stored), M3TranslationGotoProcedure.TcPOU (not stored), M3TranslationHomingProcedure.TcPOU (not stored), M3TranslationTarget.TcPOU (not stored)
//   MTCS/M3/Visu/ VISU_M3Config_General.TcVIS (not stored), VISU_M3TargetDialog.TcVIS (not stored), VISU_M3.TcVIS (not stored), VISU_M3Config.TcVIS (not stored), VISU_M3Config_KnownPosition.TcVIS (not stored), VISU_M3Config_KnownPositions.TcVIS (not stored), VISU_M3Config_Rotation_General.TcVIS (not stored), VISU_M3Config_Translation_General.TcVIS (not stored), VISU_M3Overview.TcVIS (not stored), VISU_M3Rotation.TcVIS (not stored), VISU_M3Figure.TcVIS (not stored), VISU_M3RotationDetails.TcVIS (not stored), VISU_M3RotationCurrents.TcVIS (not stored), VISU_M3TargetDialogButton.TcVIS (not stored), VISU_M3TranslationDetails.TcVIS (not stored), VISU_M3RotationFigure_1.TcVIS (not stored), VISU_M3Rotation_General.TcVIS (not stored), VISU_M3Translation.TcVIS (not stored), VISU_M3IO.TcVIS (not stored), VISU_M3Translation_General.TcVIS (not stored)
//   MTCS/M3/Widgets/ M3ConfigTabs.TcDUT (not stored), M3ConfigTabsTextList.TcTLO (not stored), M3IOWidget.TcPOU (not stored), M3RotationTabs.TcDUT (not stored), M3RotationWidget.TcPOU (not stored), M3Tabs.TcDUT (not stored), M3TargetDialogButton.TcPOU (not stored), M3TargetStatusToColor.TcPOU (not stored), M3TranslationTabs.TcDUT (not stored), M3TranslationWidget.TcPOU (not stored), M3Widget.TcPOU (not stored)
//   MTCS/MTCS/Generated/mtcs/Configs/ MTCSConfig.TcDUT (not stored), MTCSInstrumentsConfig.TcDUT (not stored)
//   MTCS/MTCS/Generated/mtcs/Processes/Args/ MTCSChangeInstrumentProcessArgs.TcDUT (not stored)
//   MTCS/MTCS/Generated/mtcs/Processes/ MTCSChangeInstrumentProcess.TcPOU (not stored)
//   MTCS/MTCS/Generated/mtcs/StateMachines/Parts/ MTCSParts.TcDUT (not stored)
//   MTCS/MTCS/Generated/mtcs/StateMachines/Processes/ MTCSProcesses.TcDUT (not stored)
//   MTCS/MTCS/Generated/mtcs/StateMachines/ SM_MTCS.TcPOU (not stored)
//   MTCS/MTCS/Generated/mtcs/StateMachines/Statuses/ MTCSStatuses.TcDUT (not stored)
//   MTCS/MTCS/ MtcsGlobalConfig.TcDUT
//   MTCS/MTCS/StateMachines/ MTCS.TcPOU
//   MTCS/MTCS/Visu/ VISU_MTCS.TcVIS (not stored), VISU_MTCSBlankScreen.TcVIS (not stored), VISU_MTCSChangeInstrumentDialog.TcVIS (not stored), VISU_MTCSParkTelescopeDialog.TcVIS (not stored), VISU_MTCSWakeUpTelescopeDialog.TcVIS (not stored), VISU_MTCSChangeOperatorDialog.TcVIS (not stored), VISU_MTCSConfigDialog.TcVIS (not stored), VISU_MTCSConfig_Instruments.TcVIS (not stored), VISU_MTCSConfig_Instrument.TcVIS (not stored), VISU_MTCSHome.TcVIS (not stored), VISU_MTCSRebootDialog.TcVIS (not stored), VISU_MTCSSidebar.TcVIS (not stored), VISU_MTCSSubSystemButton.TcVIS (not stored), VISU_MTCSSystemBackground.TcVIS (not stored), VISU_MTCSConfig.TcVIS (not stored), VISU_MTCSGoToSleepDialog.TcVIS (not stored), VISU_MTCSInitializeDialog.TcVIS (not stored)
//   MTCS/MTCS/Widgets/ MTCSChangeInstrumentDialogWidget.TcPOU (not stored), MTCSChangeOperatorDialogWidget.TcPOU (not stored), MTCSBlankScreenWidget.TcPOU (not stored), MTCSTabs.TcDUT (not stored), MTCSToColor.TcPOU (not stored), MTCSWidget.TcPOU (not stored), MTCSConfigTabsTextList.TcTLO (not stored)
//   MTCS/Safety/Generated/mtcs_safety/Configs/ SafetyConfig.TcDUT (not stored), SafetyDomeAccessAlertConfig.TcDUT (not stored), SafetyDomeAccessConfig.TcDUT (not stored)
//   MTCS/Safety/Generated/mtcs_safety/StateMachines/Parts/ SafetyDomeAccessIOParts.TcDUT (not stored), SafetyDomeAccessParts.TcDUT (not stored), SafetyHydraulicsAndSafetyIOParts.TcDUT (not stored), SafetyIOParts.TcDUT (not stored), SafetyParts.TcDUT (not stored)
//   MTCS/Safety/Generated/mtcs_safety/StateMachines/Processes/ SafetyDomeAccessProcesses.TcDUT (not stored), SafetyEmergencyStopsProcesses.TcDUT (not stored), SafetyHydraulicsProcesses.TcDUT (not stored), SafetyMotionBlockingProcesses.TcDUT (not stored), SafetyProcesses.TcDUT (not stored)
//   MTCS/Safety/Generated/mtcs_safety/StateMachines/ SM_Safety.TcPOU (not stored), SM_SafetyDomeAccess.TcPOU (not stored), SM_SafetyDomeAccessIO.TcPOU (not stored), SM_SafetyEmergencyStops.TcPOU (not stored), SM_SafetyHydraulics.TcPOU (not stored), SM_SafetyHydraulicsAndSafetyIO.TcPOU (not stored), SM_SafetyIO.TcPOU (not stored), SM_SafetyMotionBlocking.TcPOU (not stored)
//   MTCS/Safety/Generated/mtcs_safety/StateMachines/Statuses/ SafetyDomeAccessIOStatuses.TcDUT (not stored), SafetyDomeAccessStatuses.TcDUT (not stored), SafetyEmergencyStopsStatuses.TcDUT (not stored), SafetyHydraulicsAndSafetyIOStatuses.TcDUT (not stored), SafetyHydraulicsStatuses.TcDUT (not stored), SafetyIOStatuses.TcDUT (not stored), SafetyMotionBlockingStatuses.TcDUT (not stored), SafetyStatuses.TcDUT (not stored)
//   MTCS/Safety/Helper/ SafetyAlerter.TcPOU (not stored), SafetyPasswordVerifier.TcPOU (not stored)
//   MTCS/Safety/StateMachines/ SafetyHydraulicsAndSafetyIO.TcPOU (not stored), SafetyEmergencyStops.TcPOU (not stored), SafetyDomeAccess.TcPOU (not stored), SafetyDomeAccessIO.TcPOU (not stored), SafetyMotionBlocking.TcPOU (not stored), SafetyHydraulicsStates.TcDUT (not stored), SafetyIO.TcPOU (not stored), Safety.TcPOU (not stored), SafetyHydraulics.TcPOU (not stored)
//   MTCS/Safety/Visu/ VISU_Safety.TcVIS (not stored), VISU_SafetyConfig_DomeAccessGeneral.TcVIS (not stored), VISU_SafetyConfig_DomeAccessAlert.TcVIS (not stored), VISU_SafetyHydraulicsAndSafetyIO.TcVIS (not stored), VISU_SafetyEmergencyStop.TcVIS (not stored), VISU_SafetyEmergencyStops.TcVIS (not stored), VISU_SafetyDomeAccess.TcVIS (not stored), VISU_SafetyDomeAccessIO.TcVIS (not stored), VISU_SafetyMotionBlocking.TcVIS (not stored), VISU_SafetyOverview.TcVIS (not stored), VISU_SafetyIO.TcVIS (not stored), VISU_SafetyConfig.TcVIS (not stored), VISU_SafetyHydraulics.TcVIS (not stored), VISU_SafetyGroup.TcVIS (not stored)
//   MTCS/Safety/Widgets/ SafetyConfigTabsTextList.TcTLO (not stored), SafetyHydraulicsAndSafetyIOWidget.TcPOU (not stored), SafetyEmergencyStopsWidget.TcPOU (not stored), SafetyDomeAccessWidget.TcPOU (not stored), SafetyDomeAccessIOWidget.TcPOU (not stored), SafetyMotionBlockingWidget.TcPOU (not stored), SafetyIOWidget.TcPOU (not stored), SafetyTabs.TcDUT (not stored), SafetyWidget.TcPOU (not stored), SafetyHydraulicsWidget.TcPOU (not stored)
//   MTCS/Services/Generated/mtcs_services/Configs/ ServicesConfig.TcDUT (not stored), ServicesTimingConfig.TcDUT (not stored)
//   MTCS/Services/Generated/mtcs_services/Enums/ ServicesTimingPositionSource.TcDUT (not stored), ServicesTimingTimeSource.TcDUT (not stored)
//   MTCS/Services/Generated/mtcs_services/StateMachines/Parts/ ServicesParts.TcDUT (not stored), ServicesTimingIOParts.TcDUT (not stored), ServicesTimingParts.TcDUT (not stored)
//   MTCS/Services/Generated/mtcs_services/StateMachines/Processes/ ServicesProcesses.TcDUT (not stored), ServicesTimingProcesses.TcDUT (not stored)
//   MTCS/Services/Generated/mtcs_services/StateMachines/ SM_Services.TcPOU (not stored), SM_ServicesTiming.TcPOU (not stored), SM_ServicesTimingIO.TcPOU (not stored), SM_ServicesTimingSerialInfo.TcPOU (not stored)
//   MTCS/Services/Generated/mtcs_services/StateMachines/Statuses/ ServicesStatuses.TcDUT (not stored), ServicesTimingIOStatuses.TcDUT (not stored), ServicesTimingSerialInfoStatuses.TcDUT (not stored), ServicesTimingStatuses.TcDUT (not stored)
//   MTCS/Services/Helper/ TmcTimingErrorsToString.TcPOU (not stored)
//   MTCS/Services/StateMachines/ ServicesTiming.TcPOU (not stored), ServicesTimingDateTime.TcDUT (not stored), Services.TcPOU (not stored), ServicesTimingIO.TcPOU (not stored), ServicesTimingSerialInfo.TcPOU (not stored)
//   MTCS/Services/Visu/ VISU_ServicesConfig_Timing.TcVIS (not stored), VISU_ServicesTiming.TcVIS (not stored), VISU_ServicesOverview.TcVIS (not stored), VISU_ServicesConfig.TcVIS (not stored), VISU_Services.TcVIS (not stored), VISU_ServicesTimingIO.TcVIS (not stored), VISU_ServicesTimingOverview.TcVIS (not stored)
//   MTCS/Services/Widgets/ ServicesConfigTabsTextList.TcTLO (not stored), ServicesTabs.TcDUT (not stored), ServicesWidget.TcPOU (not stored), ServicesTimingIOWidget.TcPOU (not stored), ServicesTimingTabs.TcDUT (not stored), ServicesTimingWidget.TcPOU (not stored)
//   MTCS/Telemetry/Generated/mtcs_telemetry/Configs/ TelemetryAccelerometerConfig.TcDUT (not stored), TelemetryAccelerometersConfig.TcDUT (not stored), TelemetryConfig.TcDUT (not stored), TelemetryDewpointsConfig.TcDUT (not stored), TelemetryRelativeHumiditiesConfig.TcDUT (not stored), TelemetryTemperaturesConfig.TcDUT (not stored)
//   MTCS/Telemetry/Generated/mtcs_telemetry/StateMachines/Parts/ TelemetryFlatfieldLedsParts.TcDUT (not stored), TelemetryIOParts.TcDUT (not stored), TelemetryParts.TcDUT (not stored)
//   MTCS/Telemetry/Generated/mtcs_telemetry/StateMachines/Processes/ TelemetryProcesses.TcDUT (not stored)
//   MTCS/Telemetry/Generated/mtcs_telemetry/StateMachines/ SM_Telemetry.TcPOU (not stored), SM_TelemetryAccelerometer.TcPOU (not stored), SM_TelemetryAccelerometers.TcPOU (not stored), SM_TelemetryDewpoint.TcPOU (not stored), SM_TelemetryDewpoints.TcPOU (not stored), SM_TelemetryFlatfieldLeds.TcPOU (not stored), SM_TelemetryIO.TcPOU (not stored), SM_TelemetryRelativeHumidities.TcPOU (not stored), SM_TelemetryTemperatures.TcPOU (not stored)
//   MTCS/Telemetry/Generated/mtcs_telemetry/StateMachines/Statuses/ TelemetryAccelerometersStatuses.TcDUT (not stored), TelemetryAccelerometerStatuses.TcDUT (not stored), TelemetryDewpointsStatuses.TcDUT (not stored), TelemetryDewpointStatuses.TcDUT (not stored), TelemetryFlatfieldLedsStatuses.TcDUT (not stored), TelemetryIOStatuses.TcDUT (not stored), TelemetryRelativeHumiditiesStatuses.TcDUT (not stored), TelemetryStatuses.TcDUT (not stored), TelemetryTemperaturesStatuses.TcDUT (not stored)
//   MTCS/Telemetry/StateMachines/ Telemetry.TcPOU (not stored), TelemetryDewpoint.TcPOU (not stored), TelemetryDewpoints.TcPOU (not stored), TelemetryAccelerometers.TcPOU (not stored), TelemetryAccelerometer.TcPOU (not stored), TelemetryTemperatures.TcPOU (not stored), TelemetryRelativeHumidities.TcPOU (not stored), TelemetryIO.TcPOU (not stored), TelemetryFlatfieldLeds.TcPOU (not stored)
//   MTCS/Telemetry/Visu/ VISU_TelemetryAccelerometersAngles.TcVIS (not stored), VISU_TelemetryFlatfieldLeds.TcVIS (not stored), VISU_TelemetryDewpoints.TcVIS (not stored), VISU_TelemetryAccelerometers.TcVIS (not stored), VISU_TelemetryTemperatures.TcVIS (not stored), VISU_Telemetry.TcVIS (not stored), VISU_TelemetryOverview.TcVIS (not stored), VISU_TelemetryIO.TcVIS (not stored), VISU_TelemetryConfig.TcVIS (not stored), VISU_TelemetryRelativeHumidities.TcVIS (not stored)
//   MTCS/Telemetry/Widgets/ TelemetryConfigTextList.TcTLO (not stored), TelemetryAccelerometersWidget.TcPOU (not stored), TelemetryFlatfieldLedsWidget.TcPOU (not stored), TelemetryTemperaturesWidget.TcPOU (not stored), TelemetryRelativeHumiditiesWidget.TcPOU (not stored), TelemetryDewpointsWidget.TcPOU (not stored), TelemetryWidget.TcPOU (not stored), TelemetryTabs.TcDUT (not stored), TelemetryIOWidget.TcPOU (not stored)
//   POUs/ FAST.TcPOU, MAIN.TcPOU
//   VISUs/ VISU_Axes_Elevation_1_1.TcVIS (not stored), VISU_MAIN.TcVIS
// real-time tasks:
//   TASK PlcTask: cycle T#10ms, priority 14, ADS port 350
//   TASK VISU_TASK: cycle T#100000us, priority 16, ADS port 351
//   TASK PlcFastTask: cycle T#2ms, priority 8, ADS port 352
//   TASK SlalibTask: cycle T#10ms, priority 10, ADS port 353
// motion (NC):
//   TASK Fast SAF: cycle T#2ms, priority 4, ADS port 501
//   TASK NC-Task 1 SVB: cycle T#10ms, priority 12, ADS port 511
//   AXIS Cover_Top_1 (id 1)
//     General: UnitName=, IoDivider=3
//     Dynamic: AccelerationMaximum=8, DecelerationMaximum=8, Acceleration=6, Deceleration=6, Jerk=4
//     Velo: RefSearch=0, RefSync=0, SlowManual=1, FastManual=9, Maximum=9.6
//     PositionAreaControl: Range=1, RefSync=1
//     TargetPosControl: Range=0.2, Time=1
//     OtherSettings: AllowMotionCmdToSlave=true, PulseDistancePos=1, PulseDistanceNeg=1
//     encoder EncType=5
//       EncPara: ScaleFactorNumerator=360, ScaleFactorDenominator=16384, MaxCount=#x00003fff, ReferenceSystem=1
//         FilterTime: TVelo=0.2
//     drive DrvType=5
//       Analog: VeloReferenz=9.615384615
//       TimeComp: TaskDelayCycles=1
//     controller CtrType=3
//       CtrPara: PriorControlFactor=1
//         PosDiffControl: Range=15
//         PID: PosKp=5, PosTn=4
//         Observer: BandWidth=20
//   AXIS Cover_Top_2 (id 2)
//     General: UnitName=, IoDivider=3
//     Dynamic: AccelerationMaximum=8, DecelerationMaximum=8, Acceleration=6, Deceleration=6, Jerk=4
//     Velo: RefSearch=0, RefSync=0, SlowManual=1, FastManual=9, Maximum=9.6
//     PositionAreaControl: Range=1, RefSync=1
//     TargetPosControl: Range=0.2, Time=1
//     OtherSettings: AllowMotionCmdToSlave=true, PulseDistancePos=1, PulseDistanceNeg=1
//     encoder EncType=5
//       EncPara: ScaleFactorNumerator=360, ScaleFactorDenominator=16384, MaxCount=#x00003fff, ReferenceSystem=1
//         FilterTime: TVelo=0.2
//     drive DrvType=5
//       Analog: VeloReferenz=9.615384615
//       TimeComp: TaskDelayCycles=1
//     controller CtrType=3
//       CtrPara: PriorControlFactor=1
//         PosDiffControl: Range=15
//         PID: PosKp=5, PosTn=4
//         Observer: BandWidth=20
//   AXIS Cover_Top_3 (id 3)
//     General: UnitName=, IoDivider=3
//     Dynamic: AccelerationMaximum=8, DecelerationMaximum=8, Acceleration=6, Deceleration=6, Jerk=4
//     Velo: RefSearch=0, RefSync=0, SlowManual=1, FastManual=9, Maximum=9.6
//     PositionAreaControl: Range=1, RefSync=1
//     TargetPosControl: Range=0.2, Time=1
//     OtherSettings: AllowMotionCmdToSlave=true, PulseDistancePos=1, PulseDistanceNeg=1
//     encoder EncType=5
//       EncPara: ScaleFactorNumerator=360, ScaleFactorDenominator=16384, MaxCount=#x00003fff, ReferenceSystem=1
//         FilterTime: TVelo=0.2
//     drive DrvType=5
//       Analog: VeloReferenz=9.615384615
//       TimeComp: TaskDelayCycles=1
//     controller CtrType=3
//       CtrPara: PriorControlFactor=1
//         PosDiffControl: Range=15
//         PID: PosKp=7, PosTn=4
//         Observer: BandWidth=20
//   AXIS Cover_Top_4 (id 4)
//     General: UnitName=, IoDivider=3
//     Dynamic: AccelerationMaximum=8, DecelerationMaximum=8, Acceleration=6, Deceleration=6, Jerk=4
//     Velo: RefSearch=0, RefSync=0, SlowManual=1, FastManual=9, Maximum=9.6
//     PositionAreaControl: Range=1, RefSync=1
//     TargetPosControl: Range=0.2, Time=1
//     OtherSettings: AllowMotionCmdToSlave=true, PulseDistancePos=1, PulseDistanceNeg=1
//     encoder EncType=5
//       EncPara: ScaleFactorNumerator=360, ScaleFactorDenominator=16384, MaxCount=#x00003fff, ReferenceSystem=1
//         FilterTime: TVelo=0.2
//     drive DrvType=5
//       Analog: VeloReferenz=9.615384615
//       TimeComp: TaskDelayCycles=1
//     controller CtrType=3
//       CtrPara: PriorControlFactor=1
//         PosDiffControl: Range=15
//         PID: PosKp=6, PosTn=2
//         Observer: BandWidth=20
//   AXIS Cover_Bottom_1 (id 5)
//     General: UnitName=, IoDivider=3
//     Dynamic: AccelerationMaximum=8, DecelerationMaximum=8, Acceleration=6, Deceleration=6, Jerk=4
//     Velo: RefSearch=0, RefSync=0, SlowManual=1, FastManual=9, Maximum=9.6
//     PositionAreaControl: Range=1, RefSync=1
//     TargetPosControl: Range=0.2, Time=1
//     OtherSettings: AllowMotionCmdToSlave=true, PulseDistancePos=1, PulseDistanceNeg=1
//     encoder EncType=5
//       EncPara: ScaleFactorNumerator=360, ScaleFactorDenominator=16384, MaxCount=#x00003fff, ReferenceSystem=1
//         FilterTime: TVelo=0.2
//     drive DrvType=5
//       Analog: VeloReferenz=9.615384615
//       TimeComp: TaskDelayCycles=1
//     controller CtrType=3
//       CtrPara: PriorControlFactor=1
//         PosDiffControl: Range=15
//         PID: PosKp=5, PosTn=4
//         Observer: BandWidth=20
//   AXIS Cover_Bottom_2 (id 6)
//     General: UnitName=, IoDivider=3
//     Dynamic: AccelerationMaximum=8, DecelerationMaximum=8, Acceleration=6, Deceleration=6, Jerk=4
//     Velo: RefSearch=0, RefSync=0, SlowManual=1, FastManual=9, Maximum=9.6
//     PositionAreaControl: Range=1, RefSync=1
//     TargetPosControl: Range=0.2, Time=1
//     OtherSettings: AllowMotionCmdToSlave=true, PulseDistancePos=1, PulseDistanceNeg=1
//     encoder EncType=5
//       EncPara: ScaleFactorNumerator=360, ScaleFactorDenominator=16384, MaxCount=#x00003fff, ReferenceSystem=1
//         FilterTime: TVelo=0.2
//     drive DrvType=5
//       Analog: VeloReferenz=9.615384615
//       TimeComp: TaskDelayCycles=1
//     controller CtrType=3
//       CtrPara: PriorControlFactor=1
//         PosDiffControl: Range=15
//         PID: PosKp=5, PosTn=4
//         Observer: BandWidth=20
//   AXIS Cover_Bottom_3 (id 7)
//     General: UnitName=, IoDivider=3
//     Dynamic: AccelerationMaximum=8, DecelerationMaximum=8, Acceleration=6, Deceleration=6, Jerk=4
//     Velo: RefSearch=0, RefSync=0, SlowManual=1, FastManual=9, Maximum=9.6
//     PositionAreaControl: Range=1, RefSync=1
//     TargetPosControl: Range=0.2, Time=1
//     OtherSettings: AllowMotionCmdToSlave=true, PulseDistancePos=1, PulseDistanceNeg=1
//     encoder EncType=5
//       EncPara: ScaleFactorNumerator=360, ScaleFactorDenominator=16384, MaxCount=#x00003fff, ReferenceSystem=1
//         FilterTime: TVelo=0.2
//     drive DrvType=5
//       Analog: VeloReferenz=9.615384615
//       TimeComp: TaskDelayCycles=1
//     controller CtrType=3
//       CtrPara: PriorControlFactor=1
//         PosDiffControl: Range=15
//         PID: PosKp=5, PosTn=2
//         Observer: BandWidth=20
//   AXIS Cover_Bottom_4 (id 8)
//     General: UnitName=, IoDivider=3
//     Dynamic: AccelerationMaximum=8, DecelerationMaximum=8, Acceleration=6, Deceleration=6, Jerk=4
//     Velo: RefSearch=0, RefSync=0, SlowManual=1, FastManual=9, Maximum=9.6
//     PositionAreaControl: Range=1, RefSync=1
//     TargetPosControl: Range=0.2, Time=1
//     OtherSettings: AllowMotionCmdToSlave=true, PulseDistancePos=1, PulseDistanceNeg=1
//     encoder EncType=5
//       EncPara: ScaleFactorNumerator=360, ScaleFactorDenominator=16384, MaxCount=#x00003fff, ReferenceSystem=1
//         FilterTime: TVelo=0.2
//     drive DrvType=5
//       Analog: VeloReferenz=9.615384615
//       TimeComp: TaskDelayCycles=1
//     controller CtrType=3
//       CtrPara: PriorControlFactor=1
//         PosDiffControl: Range=15
//         PID: PosKp=4, PosTn=5
//         Observer: BandWidth=20
//   AXIS M3_RotationPositioning (id 9)
//     General: UnitName=°, IoDivider=3
//     Dynamic: AccelerationMaximum=3, DecelerationMaximum=3, Acceleration=2.8, Deceleration=2.8, Jerk=2.8
//     Velo: RefSearch=1, RefSync=1, SlowManual=0.3, FastManual=2.5, Maximum=2.8
//     PositionAreaControl: Enable=false, RefSearch=false
//     TargetPosControl: Range=0.03
//     OtherSettings: AllowMotionCmdToSlave=true, PulseDistancePos=0.5, PulseDistanceNeg=0.5
//     encoder EncType=5
//       EncPara: ScaleFactorNumerator=360, ScaleFactorDenominator=786432, ReferenceSystem=1
//     drive DrvType=16
//       DrvPara: MaxCount=#xffffffff
//         Analog: VeloReferenz=2.7
//         TimeComp: TaskDelayCycles=1
//     controller CtrType=1
//       CtrPara: PriorControlFactor=1
//         PosDiffControl: Range=10
//         PID: CtrlOutputLimit=1
//         Observer: BandWidth=20
//   AXIS M3_Translation (id 11)
//     General: IoDivider=3
//     Dynamic: AccelerationMaximum=2, DecelerationMaximum=2, Acceleration=2, Deceleration=2, Jerk=3
//     Velo: RefSearch=0.5, RefSync=0.5, SlowManual=0.1, FastManual=1.5, Fast=1.5, Maximum=1.55039
//     PositionAreaControl: Enable=false, RefSearch=false
//     TargetPosControl: Enable=false
//     OtherSettings: AllowMotionCmdToSlave=true, PulseDistancePos=0.3, PulseDistanceNeg=0.3
//     encoder EncType=4
//       EncPara: ScaleFactorNumerator=5e-005, MaxCount=#x0000ffff
//         FilterTime: TVelo=0.2
//         Inc: RefMode=2, RefSoftSyncMask=#x0000ffff
//     drive DrvType=16
//       DrvPara: MaxCount=#xffffffff
//         Analog: VeloReferenz=1.55039, VeloScale=2.5
//         TimeComp: TaskDelayCycles=1
//     controller CtrType=1
//       CtrPara: PriorControlFactor=1
//         PosDiffControl: Enable=false
//         Observer: BandWidth=20
//   AXIS M3_RotationAntiBacklash (id 10)
//     General: UnitName=°, IoDivider=3
//     Dynamic: AccelerationMaximum=20, DecelerationMaximum=20, Acceleration=16.8, Deceleration=16.8, Jerk=16.8
//     Velo: RefSearch=5, RefSync=5, SlowManual=1, FastManual=15, Maximum=16.8
//     PositionAreaControl: Enable=false, RefSearch=false
//     TargetPosControl: Enable=false
//     OtherSettings: AllowMotionCmdToSlave=true, PulseDistancePos=2, PulseDistanceNeg=2
//     encoder EncType=19
//       EncPara: ScaleFactorNumerator=360, ScaleFactorDenominator=4800000, MaxCount=#xffffffff
//     drive DrvType=16
//       DrvPara: MaxCount=#xffffffff
//         Analog: VeloReferenz=16.2, VeloScale=2.5
//         TimeComp: TaskDelayCycles=1
//     controller CtrType=1
//       CtrPara: PriorControlFactor=1
//         PosDiffControl: Enable=false, Range=50
//         PID: PosKp=5
//         Observer: BandWidth=20
//   AXIS M3_RotationPosHall (id 12)
//     General: UnitName=°, IoDivider=3
//     OtherSettings: AllowMotionCmdToSlave=true
//     encoder EncType=19
//       EncPara: ScaleFactorNumerator=360, ScaleFactorDenominator=4800000, MaxCount=#xffffffff
//         FilterTime: TVelo=0.2
//     drive DrvType=5
//       TimeComp: TaskDelayCycles=1
//     controller CtrType=1
//       CtrPara: PriorControlFactor=1
//         Observer: BandWidth=20
//   AXIS AZI_Virtual (id 18)
//     General: UnitName=°
//     Dynamic: AccelerationMaximum=3, DecelerationMaximum=5, Acceleration=1.5, Deceleration=1.5, Jerk=2.3
//     Velo: SlowManual=0.1, FastManual=3, Maximum=3.2
//     OtherSettings: AllowMotionCmdToSlave=true
//     encoder EncType=1
//       SoftEndMaxControl: Enable=true, Range=370
//     drive DrvType=5
//       Analog: VeloReferenz=3
//     controller CtrType=1
//       CtrPara: PriorControlFactor=1
//         Observer: BandWidth=20
//   AXIS AZI_Physical (id 13) // Azimuth driving axis (i.e. not the anti-backlash axis)
//     General: UnitName=°
//     Dynamic: AccelerationMaximum=3, DecelerationMaximum=5, Acceleration=1.5, Deceleration=1.5, Jerk=2.3
//     Velo: RefSearch=1, RefSync=1, SlowManual=0.1, FastManual=1, Fast=3288.14869333333, Maximum=3.2
//     OtherSettings: AllowMotionCmdToSlave=true, AllowMotionCmdToExtSetGenAxis=true, PulseDistancePos=0.1, PulseDistanceNeg=0.1
//     encoder EncType=8
//       EncPara: ScaleFactorNumerator=360, ScaleFactorDenominator=1509949440, MaxCount=#xffffffff
//         FilterTime: TVelo=0.05
//         SoftEndMinControl: Range=-5
//         SoftEndMaxControl: Range=370
//         ActPosCorrection: Enable=true, Time=0.05
//     drive DrvType=9
//       DrvPara: MaxCount=#xffffffff, DriveControlDWord=#x00030100
//         Analog: VeloReferenz=3, VeloScale=1.02400649589962
//         TimeComp: TaskDelayCycles=1
//     controller CtrType=1
//       CtrPara: PriorControlFactor=1
//         PID: PosKp=0.1
//         Observer: BandWidth=20
//   AXIS AZI_ABL (id 14) // Azimuth Anti-Backlash axis
//     General: UnitName=°
//     Dynamic: AccelerationMaximum=3, DecelerationMaximum=5, Acceleration=1.5, Deceleration=1.5, Jerk=2.3
//     Velo: RefSearch=1, RefSync=1, SlowManual=0.1, FastManual=1, Maximum=3.2
//     PositionAreaControl: Enable=false, RefSearch=false
//     TargetPosControl: Enable=false
//     OtherSettings: AllowMotionCmdToSlave=true, PulseDistancePos=0.1, PulseDistanceNeg=0.1
//     encoder EncType=8
//       EncPara: ScaleFactorNumerator=360, ScaleFactorDenominator=188743680, MaxCount=#xffffffff
//     drive DrvType=9
//       DrvPara: MaxCount=#xffffffff
//         Analog: VeloReferenz=3, VeloScale=1.02400649589962
//         TimeComp: TaskDelayCycles=1
//     controller CtrType=1
//       CtrPara: PriorControlFactor=1
//         PosDiffControl: Enable=false
//         Observer: BandWidth=20
//   AXIS ELE_Virtual (id 19)
//     General: UnitName=°
//     Dynamic: AccelerationMaximum=3, DecelerationMaximum=5, Acceleration=1.5, Deceleration=1.5, Jerk=2.3
//     Velo: RefSearch=1, RefSync=1, SlowManual=0.1, FastManual=3, Maximum=3.2
//     OtherSettings: AllowMotionCmdToSlave=true, PulseDistancePos=0.1, PulseDistanceNeg=0.1
//     encoder EncType=1
//     drive DrvType=5
//       Analog: VeloReferenz=3
//     controller CtrType=1
//       CtrPara: PriorControlFactor=1
//         Observer: BandWidth=20
//   AXIS ELE_Physical (id 15) // Elevation axis
//     General: UnitName=°
//     Dynamic: AccelerationMaximum=3, DecelerationMaximum=5, Acceleration=1.5, Deceleration=1.5, Jerk=2.3
//     Velo: RefSearch=1, RefSync=1, SlowManual=0.1, FastManual=1, Fast=11288.9626464844, Maximum=3.2
//     OtherSettings: AllowMotionCmdToSlave=true, PulseDistancePos=0.1, PulseDistanceNeg=0.1
//     encoder EncType=8
//       EncPara: ScaleFactorNumerator=360, ScaleFactorDenominator=1509949440, MaxCount=#xffffffff
//     drive DrvType=9
//       DrvPara: MaxCount=#xffffffff, DriveControlDWord=#x00030100
//         Analog: VeloReferenz=3, VeloScale=1.02400649589962
//         TimeComp: TaskDelayCycles=1
//     controller CtrType=1
//       CtrPara: PriorControlFactor=1
//         Observer: BandWidth=20
//   AXIS ROC_Virtual (id 20)
//     Dynamic: AccelerationMaximum=6, DecelerationMaximum=13, Acceleration=3, Deceleration=3, Jerk=5
//     Velo: RefSearch=3, RefSync=3, SlowManual=1, FastManual=6, Maximum=6.2
//     OtherSettings: AllowMotionCmdToSlave=true, PulseDistancePos=1, PulseDistanceNeg=1
//     encoder EncType=1
//       EncPara: ScaleFactorNumerator=360, ScaleFactorDenominator=1073741824
//     drive DrvType=5
//       Analog: VeloReferenz=6
//     controller CtrType=1
//       CtrPara: PriorControlFactor=1
//         Observer: BandWidth=20
//   AXIS ROC_Physical (id 16) // deROtator for Cassegrain
//     General: UnitName=°
//     Dynamic: AccelerationMaximum=6, DecelerationMaximum=13, Acceleration=3, Deceleration=3, Jerk=5
//     Velo: RefSearch=3, RefSync=3, SlowManual=0.2, FastManual=2, Fast=18000, Maximum=6.3
//     OtherSettings: AllowMotionCmdToSlave=true, PulseDistancePos=0.2, PulseDistanceNeg=0.2
//     encoder EncType=8
//       EncPara: ScaleFactorNumerator=360, ScaleFactorDenominator=1073741824, Offset=-54.2229, MaxCount=#xffffffff
//     drive DrvType=9
//       DrvPara: MaxCount=#xffffffff, DriveControlDWord=#x00030100
//         Analog: VeloReferenz=6, VeloScale=1.02400649589962
//         TimeComp: TaskDelayCycles=1
//     controller CtrType=1
//       CtrPara: PriorControlFactor=1
//         Observer: BandWidth=20
//   AXIS RON_Physical (id 17) // deROtator for Nasmyth
//     General: UnitName=°
//     Dynamic: AccelerationMaximum=6, DecelerationMaximum=13, Acceleration=3, Deceleration=3, Jerk=5
//     Velo: RefSearch=3, RefSync=3, SlowManual=0.2, FastManual=2, Maximum=6.3
//     OtherSettings: AllowMotionCmdToSlave=true, PulseDistancePos=0.2, PulseDistanceNeg=0.2
//     encoder EncType=8
//       EncPara: ScaleFactorNumerator=360, ScaleFactorDenominator=1073741824, Offset=-51.6118, MaxCount=#xffffffff
//     drive DrvType=9
//       DrvPara: MaxCount=#xffffffff, DriveControlDWord=#x00030100
//         Analog: VeloReferenz=6, VeloScale=1.02400649589962
//         TimeComp: TaskDelayCycles=1
//     controller CtrType=1
//       CtrPara: PriorControlFactor=1
//         Observer: BandWidth=20
//   AXIS RON_Virtual (id 21)
//     Dynamic: AccelerationMaximum=6, DecelerationMaximum=13, Acceleration=3, Deceleration=3, Jerk=5
//     Velo: RefSearch=3, RefSync=3, SlowManual=0.2, FastManual=2, Maximum=6.2
//     OtherSettings: AllowMotionCmdToSlave=true, PulseDistancePos=0.2, PulseDistanceNeg=0.2
//     encoder EncType=1
//     drive DrvType=5
//       Analog: VeloReferenz=6
//     controller CtrType=1
//       CtrPara: PriorControlFactor=1
//         Observer: BandWidth=20
//   AXIS FW_Physical (id 22)
//     General: UnitName=°
//     OtherSettings: AllowMotionCmdToSlave=true
//     encoder EncType=8
//       EncPara: MaxCount=#xffffffff
//     drive DrvType=9
//       DrvPara: MaxCount=#xffffffff, DriveControlDWord=#x00000100
//         Analog: VeloScale=1.02400649589962
//         TimeComp: TaskDelayCycles=1
//     controller CtrType=1
//       CtrPara: PriorControlFactor=1
//         Observer: BandWidth=20
// I/O:
//   DEVICE ECAT (EtherCAT), AmsNetId 161.72.58.86.3.1
//     Pumps room star point - coupler (EK1101) [EK1101 EtherCAT Coupler (2A E-Bus, ID switch)]
//       Pumps room star point - Slot 1 (EK1122) [EK1122 2 port EtherCAT junction]
//         Timing coupler (EK1100) [EK1100 EtherCAT Coupler (2A E-Bus)]
//           Timing Slot 1 (serial EL6001) [EL6001 Interface (RS232)]
//           Timing Slot 2 (PTP EL6688) [EL6688 - External Synchronisation Interface (IEEE1588)]
//           Timing End cap (EL9011) [EL9011 End Terminal]
//         REM star point (CU1128) [CU1128 6x EtherCAT junction]
//           Cover coupler (EK1101) [EK1101 EtherCAT Coupler (2A E-Bus, ID switch)]
//             Cover slot 1 (digital out, EL2008) [EL2008 8Ch. Dig. Output 24V, 0.5A]
//             Cover slot 2 (analog out, EL4008) [EL4008 8Ch. Ana. Output 0-10V, 12bit]
//             Cover slot 3 (digital in, EL1088) [EL1088 8Ch. Dig. Input 24V, 3ms, negative]
//             Cover slot 4 (enc top 1-2, EL5002) [EL5002 2Ch. SSI Encoder]
//             Cover slot 5 (enc top 3-4, EL5002) [EL5002 2Ch. SSI Encoder]
//             Cover slot 6 (enc bot 1-2, EL5002) [EL5002 2Ch. SSI Encoder]
//             Cover slot 7 (enc bot 3-4, EL5002) [EL5002 2Ch. SSI Encoder]
//             Cover slot 8 (relays top 1-2, EL2622) [EL2622 2Ch. Relay Output, NO (230V AC / 30V DC)]
//             Cover slot 9 (relays top 3-4, EL2622) [EL2622 2Ch. Relay Output, NO (230V AC / 30V DC)]
//             Cover slot 10 (relays bot 1-2, EL2622) [EL2622 2Ch. Relay Output, NO (230V AC / 30V DC)]
//             Cover slot 11 (relays bot 3-4, EL2622) [EL2622 2Ch. Relay Output, NO (230V AC / 30V DC)]
//             Cover slot 12 (relays magnet top-bot, EL2622) [EL2622 2Ch. Relay Output, NO (230V AC / 30V DC)]
//             Cover slot 13 (multimeter, EL3681) [EL3681 Digital multimeter terminal]
//             Cover end cap (EL9011) [EL9011 End Terminal]
//           M1M2:COU (EK1101) [EK1101 EtherCAT Coupler (2A E-Bus, ID switch)]
//             M1M2:AI1 (Analog in, EL3102) [EL3102 2Ch. Ana. Input +/-10V, Diff.]
//             M1M2:AI2 (Analog in, EL3024) [EL3024 4Ch. Ana. Input 4-20mA DIFF]
//             M1M2:AI3 (Analog in, EL3024) [EL3024 4Ch. Ana. Input 4-20mA DIFF]
//             M1M2:AO1 (Analog out, EL4022) [EL4022 2Ch. Ana. Output 4-20mA, 12bit]
//             M1M2:DO1 (Digital out, EL2024) [EL2024 4Ch. Dig. Output 24V, 2A]
//             M1M2:RES1 (Res bridge SO, EL3351) [EL3351 1Ch. Ana. Input Resistor Bridge Terminal, Diff. 16bit]
//             M1M2:RES2 (Res bridge NE, EL3351) [EL3351 1Ch. Ana. Input Resistor Bridge Terminal, Diff. 16bit]
//             M1M2:RES3 (Res bridge NW, EL3351) [EL3351 1Ch. Ana. Input Resistor Bridge Terminal, Diff. 16bit]
//             M1M2:PWR1 (Power supply, EL9410) [EL9410 E-Bus Power Supplier  (Diagnostics)]
//             M1M2:SSI1 (SSI encoder, EL5001) [EL5001 1Ch. SSI Encoder]
//             M1M2:AI4 (Analog in, EL3164) [EL3164 4Ch. Ana. Input 0-10V]
//             M1M2:INC1 (Counter, EL5101) [EL5101 1Ch. Inc. Encoder 5V]
//             M1M2:5V1 (Power 5V, EL9505) [EL9505 Power supply terminal 5V]
//             M1M2:DO2 (Digital out, EL2124) [EL2124 4Ch. Dig. Output 5V, 20mA]
//             M1M2:DO3 (Digital out, EL2124) [EL2124 4Ch. Dig. Output 5V, 20mA]
//             M1M2:RE1 (Relay, EL2622) [EL2622 2Ch. Relay Output, NO (230V AC / 30V DC)]
//             M1M2:END (EL9011) [EL9011 End Terminal]
//           REM star point B (CU1128-B) [CU1128 6x EtherCAT junction - Dev A]
//             M3 coupler (EK1100) [EK1100 EtherCAT Coupler (2A E-Bus)]
//               M3 Slot 1 (digital in EL1088) [EL1088 8Ch. Dig. Input 24V, 3ms, negative]
//               M3 Slot 2 (encoder EL5101) [EL5101 1Ch. Inc. Encoder 5V]
//               M3 Slot 3 (encoder EL5001) [EL5001 1Ch. SSI Encoder]
//               M3 Slot 4 (CANopen EL6751) [EL6751 CANopen Master]
//               M3 End cap (EL9011) [EL9011 End Terminal]
//             Accelerometer box (EP1816-3008) [EP1816-3008 16Ch. Dig. Input  24V 10µs Acceleration Sensor, DSUB-25]
//             Telemetry coupler (EK1101) [EK1101 EtherCAT Coupler (2A E-Bus, ID switch)]
//               Slot 5 (EL3202-0010) [EL3202-0010 2Ch. Ana. Input PT100 (RTD), High Precision]
//               Slot 6 (EL3202-0010) [EL3202-0010 2Ch. Ana. Input PT100 (RTD), High Precision]
//               Slot 7 (EL3202-0010) [EL3202-0010 2Ch. Ana. Input PT100 (RTD), High Precision]
//               Slot 8 (EL3202-0010) [EL3202-0010 2Ch. Ana. Input PT100 (RTD), High Precision]
//               Slot 9 (EL3202-0010) [EL3202-0010 2Ch. Ana. Input PT100 (RTD), High Precision]
//               Slot 10 (EL3202-0010) [EL3202-0010 2Ch. Ana. Input PT100 (RTD), High Precision]
//               Slot 11 (EL3202-0010) [EL3202-0010 2Ch. Ana. Input PT100 (RTD), High Precision]
//               Slot 12 (EL3024) [EL3024 4Ch. Ana. Input 4-20mA DIFF]
//               Slot 13 (EL2008) [EL2008 8Ch. Dig. Output 24V, 0.5A]
//               Term 58 (EL9011) [EL9011 End Terminal]
//           REM star point C (CU1128-C) [CU1128 6x EtherCAT junction - Dev B]
//             TE:COU (EK1101) [EK1101 EtherCAT Coupler (2A E-Bus, ID switch)] // Telescope Encoders coupler
//               TE:EN1 (EL5101) [EL5101 1Ch. Inc. Encoder 5V]
//               TE:EN2 (EL5101) [EL5101 1Ch. Inc. Encoder 5V]
//               TE:EN3 (EL5101) [EL5101 1Ch. Inc. Encoder 5V]
//               TE:EN4 (EL5101) [EL5101 1Ch. Inc. Encoder 5V]
//               TE:EN5 (EL5101) [EL5101 1Ch. Inc. Encoder 5V]
//               TE:EN6 (EL5101) [EL5101 1Ch. Inc. Encoder 5V]
//               TE:EN7 (EL5002) [EL5002 2Ch. SSI Encoder]
//               TE:END (EL9011) [EL9011 End Terminal]
//             AZID (AX5206-0000-0203) [AX5206-0000-0203 EtherCAT Drive (SoE, 2 Ch.)]
//               AZID:SAFE (AX5805) [AX5805 (Safety Drive Option)]
//                 modules: Module 1 (Safety Process Data, 2 axis), Module 2 (Standard Process Data, 2 axis)
//               AZID:END (EL9011) [EL9011 End Terminal]
//             ABLD (AX5206-0000-0203) [AX5206-0000-0203 EtherCAT Drive (SoE, 2 Ch.)]
//               ABLD:SAFE (AX5805) [AX5805 (Safety Drive Option)]
//                 modules: Module 1 (Safety Process Data, 2 axis), Module 2 (Standard Process Data, 2 axis)
//               ABLD:END (EL9011) [EL9011 End Terminal]
//             ELED (AX5206-0000-0203) [AX5206-0000-0203 EtherCAT Drive (SoE, 2 Ch.)]
//               ELED:SAFE (AX5805) [AX5805 (Safety Drive Option)]
//                 modules: Module 1 (Safety Process Data, 2 axis), Module 2 (Standard Process Data, 2 axis)
//               ELED:END (EL9011) [EL9011 End Terminal]
//       Pumps room star point - Slot 2 (EK1122) [EK1122 2 port EtherCAT junction]
//         HS: Hydraulics & Safety [EK1101 EtherCAT Coupler (2A E-Bus, ID switch)]
//           HS:DO1 (EL2008) [EL2008 8Ch. Dig. Output 24V, 0.5A]
//           HS:SI1 (EL1904) [EL1904, 4 Ch. Safety Input 24V, TwinSAFE]
//             modules: Module 1 (FSOES)
//           HS:SI2 (EL1904) [EL1904, 4 Ch. Safety Input 24V, TwinSAFE]
//             modules: Module 1 (FSOES)
//           HS:SI3 (EL1904) [EL1904, 4 Ch. Safety Input 24V, TwinSAFE]
//             modules: Module 1 (FSOES)
//           HS:SI4 (EL1904) [EL1904, 4 Ch. Safety Input 24V, TwinSAFE]
//             modules: Module 1 (FSOES)
//           HS:SL (EL6900) [EL6900, TwinSAFE PLC]
//           HS:SO1 (EL2904) [EL2904, 4 Ch. Safety Output 24V, 0.5A, TwinSAFE]
//             modules: Module 1 (FSOES), Module 2 (DO)
//           HS:AI1 (EL3102) [EL3102 2Ch. Ana. Input +/-10V, Diff.]
//           HS:AI2 (EL3152) [EL3152 2Ch. Ana Input 4-20mA]
//           HS:RTD1 (EL3202-0010) [EL3202-0010 2Ch. Ana. Input PT100 (RTD), High Precision]
//           HS:PWR1 (EL9410) [EL9410 E-Bus Power Supplier  (Diagnostics)]
//           HS:AO1 (EL4132) [EL4132 2Ch. Ana. Output +/-10V, 16bit]
//           HS:END (EL9011) [EL9011 End Terminal]
//         PG: Pumps Group [EK1101 EtherCAT Coupler (2A E-Bus, ID switch)]
//           PG:DI1 (EL1008) [EL1008 8Ch. Dig. Input 24V, 3ms]
//           PG:SI1 (EL1904) [EL1904, 4 Ch. Safety Input 24V, TwinSAFE]
//             modules: Module 1 (FSOES)
//           PG:SI2 (EL1904) [EL1904, 4 Ch. Safety Input 24V, TwinSAFE]
//             modules: Module 1 (FSOES)
//           PG:SI3 (EL1904) [EL1904, 4 Ch. Safety Input 24V, TwinSAFE]
//             modules: Module 1 (FSOES)
//           PG:DI2 (EL1008) [EL1008 8Ch. Dig. Input 24V, 3ms]
//           PG:END (EL9011) [EL9011 End Terminal]
//       Pumps room star point - Slot 3 (EK1122) [EK1122 2 port EtherCAT junction]
//         DA: Dome Access [EK1101 EtherCAT Coupler (2A E-Bus, ID switch)]
//           DA:DI1 (EL1008) [EL1008 8Ch. Dig. Input 24V, 3ms]
//           DA:DI2 (EL1008) [EL1008 8Ch. Dig. Input 24V, 3ms]
//           DA:DO1 (EL2008) [EL2008 8Ch. Dig. Output 24V, 0.5A]
//           DA:SI1 (EL1904) [EL1904, 4 Ch. Safety Input 24V, TwinSAFE]
//             modules: Module 1 (FSOES)
//           DA:RE1 (EL2622) [EL2622 2Ch. Relay Output, NO (230V AC / 30V DC)]
//           DA:RE2 (EL2622) [EL2622 2Ch. Relay Output, NO (230V AC / 30V DC)]
//           DA:END (EL9011) [EL9011 End Terminal]
//   DEVICE M3 CANopen bus, AmsNetId 161.72.58.86.2.1
//     Box 1 (MCBL3006S-CO) - LINMOT
//     Box 2 (MCBL3006S-CO) - ROTPOS
//     Box 3 (MCBL3006S-CO) - ROTABL
// variable links:
//   ECAT (EtherCAT) <-> ECAT (EtherCAT)/Pumps room star point - coupler (EK1101)/Pumps room star point - Slot 1 (EK1122)/REM star point (CU1128)/REM star point C (CU1128-C)/ABLD (AX5206-0000-0203)/ABLD:SAFE (AX5805)
//     Pumps room star point - coupler (EK1101)/Pumps room star point - Slot 2 (EK1122)/HS: Hydraulics & Safety/HS:SL (EL6900)/ConnectionInputs/Message_94 TxPDO <-> Module 1 (Safety Process Data, 2 axis)/Outputs (Controlword)/FSOE
//   ECAT (EtherCAT) <-> ECAT (EtherCAT)/Pumps room star point - coupler (EK1101)/Pumps room star point - Slot 1 (EK1122)/REM star point (CU1128)/REM star point C (CU1128-C)/AZID (AX5206-0000-0203)/AZID:SAFE (AX5805)
//     Pumps room star point - coupler (EK1101)/Pumps room star point - Slot 2 (EK1122)/HS: Hydraulics & Safety/HS:SL (EL6900)/ConnectionOutputs/Message_93 RxPDO <-> Module 1 (Safety Process Data, 2 axis)/Inputs (Statusword)/FSOE
//   ECAT (EtherCAT) <-> ECAT (EtherCAT)/Pumps room star point - coupler (EK1101)/Pumps room star point - Slot 1 (EK1122)/REM star point (CU1128)/REM star point C (CU1128-C)/ELED (AX5206-0000-0203)/ELED:SAFE (AX5805)
//     Pumps room star point - coupler (EK1101)/Pumps room star point - Slot 2 (EK1122)/HS: Hydraulics & Safety/HS:SL (EL6900)/ConnectionInputs/Message_95 TxPDO <-> Module 1 (Safety Process Data, 2 axis)/Outputs (Controlword)/FSOE
//   ECAT (EtherCAT) <-> ECAT (EtherCAT)/Pumps room star point - coupler (EK1101)/Pumps room star point - Slot 2 (EK1122)/HS: Hydraulics & Safety/HS:SI1 (EL1904)
//     Pumps room star point - coupler (EK1101)/Pumps room star point - Slot 2 (EK1122)/HS: Hydraulics & Safety/HS:SL (EL6900)/ConnectionOutputs/Message_76 RxPDO <-> Module 1 (FSOES)/TxPDO/FSOE
//   ECAT (EtherCAT) <-> ECAT (EtherCAT)/Pumps room star point - coupler (EK1101)/Pumps room star point - Slot 2 (EK1122)/HS: Hydraulics & Safety/HS:SI2 (EL1904)
//     Pumps room star point - coupler (EK1101)/Pumps room star point - Slot 2 (EK1122)/HS: Hydraulics & Safety/HS:SL (EL6900)/ConnectionInputs/Message_77 TxPDO <-> Module 1 (FSOES)/RxPDO/FSOE
//     Pumps room star point - coupler (EK1101)/Pumps room star point - Slot 2 (EK1122)/HS: Hydraulics & Safety/HS:SL (EL6900)/ConnectionOutputs/Message_77 RxPDO <-> Module 1 (FSOES)/TxPDO/FSOE
//   ECAT (EtherCAT) <-> ECAT (EtherCAT)/Pumps room star point - coupler (EK1101)/Pumps room star point - Slot 2 (EK1122)/HS: Hydraulics & Safety/HS:SI3 (EL1904)
//     Pumps room star point - coupler (EK1101)/Pumps room star point - Slot 2 (EK1122)/HS: Hydraulics & Safety/HS:SL (EL6900)/ConnectionInputs/Message_73 TxPDO <-> Module 1 (FSOES)/RxPDO/FSOE
//   ECAT (EtherCAT) <-> ECAT (EtherCAT)/Pumps room star point - coupler (EK1101)/Pumps room star point - Slot 2 (EK1122)/HS: Hydraulics & Safety/HS:SI4 (EL1904)
//     Pumps room star point - coupler (EK1101)/Pumps room star point - Slot 2 (EK1122)/HS: Hydraulics & Safety/HS:SL (EL6900)/ConnectionOutputs/Message_75 RxPDO <-> Module 1 (FSOES)/TxPDO/FSOE
//   ECAT (EtherCAT) <-> ECAT (EtherCAT)/Pumps room star point - coupler (EK1101)/Pumps room star point - Slot 2 (EK1122)/HS: Hydraulics & Safety/HS:SL (EL6900)
//     Pumps room star point - coupler (EK1101)/Pumps room star point - Slot 1 (EK1122)/REM star point (CU1128)/REM star point C (CU1128-C)/ABLD (AX5206-0000-0203)/ABLD:SAFE (AX5805)/Module 1 (Safety Process Data, 2 axis)/Inputs (Statusword)/FSOE <-> ConnectionOutputs/Message_94 RxPDO
//     Pumps room star point - coupler (EK1101)/Pumps room star point - Slot 1 (EK1122)/REM star point (CU1128)/REM star point C (CU1128-C)/AZID (AX5206-0000-0203)/AZID:SAFE (AX5805)/Module 1 (Safety Process Data, 2 axis)/Outputs (Controlword)/FSOE <-> ConnectionInputs/Message_93 TxPDO
//     Pumps room star point - coupler (EK1101)/Pumps room star point - Slot 1 (EK1122)/REM star point (CU1128)/REM star point C (CU1128-C)/ELED (AX5206-0000-0203)/ELED:SAFE (AX5805)/Module 1 (Safety Process Data, 2 axis)/Inputs (Statusword)/FSOE <-> ConnectionOutputs/Message_95 RxPDO
//     Pumps room star point - coupler (EK1101)/Pumps room star point - Slot 2 (EK1122)/HS: Hydraulics & Safety/HS:SI1 (EL1904)/Module 1 (FSOES)/RxPDO/FSOE <-> ConnectionInputs/Message_76 TxPDO
//     Pumps room star point - coupler (EK1101)/Pumps room star point - Slot 2 (EK1122)/HS: Hydraulics & Safety/HS:SI4 (EL1904)/Module 1 (FSOES)/RxPDO/FSOE <-> ConnectionInputs/Message_75 TxPDO
//     Pumps room star point - coupler (EK1101)/Pumps room star point - Slot 2 (EK1122)/HS: Hydraulics & Safety/HS:SI3 (EL1904)/Module 1 (FSOES)/TxPDO/FSOE <-> ConnectionOutputs/Message_73 RxPDO
//     Pumps room star point - coupler (EK1101)/Pumps room star point - Slot 2 (EK1122)/HS: Hydraulics & Safety/HS:SO1 (EL2904)/Module 1 (FSOES)/TxPDO/FSOE <-> ConnectionOutputs/Message_91 RxPDO
//     Pumps room star point - coupler (EK1101)/Pumps room star point - Slot 2 (EK1122)/PG: Pumps Group/PG:SI1 (EL1904)/Module 1 (FSOES)/TxPDO/FSOE <-> ConnectionOutputs/Message_78 RxPDO
//     Pumps room star point - coupler (EK1101)/Pumps room star point - Slot 2 (EK1122)/PG: Pumps Group/PG:SI2 (EL1904)/Module 1 (FSOES)/TxPDO/FSOE <-> ConnectionOutputs/Message_79 RxPDO
//     Pumps room star point - coupler (EK1101)/Pumps room star point - Slot 2 (EK1122)/PG: Pumps Group/PG:SI3 (EL1904)/Module 1 (FSOES)/TxPDO/FSOE <-> ConnectionOutputs/Message_80 RxPDO
//     Pumps room star point - coupler (EK1101)/Pumps room star point - Slot 3 (EK1122)/DA: Dome Access/DA:SI1 (EL1904)/Module 1 (FSOES)/TxPDO/FSOE <-> ConnectionOutputs/Message_84 RxPDO
//   ECAT (EtherCAT) <-> ECAT (EtherCAT)/Pumps room star point - coupler (EK1101)/Pumps room star point - Slot 2 (EK1122)/HS: Hydraulics & Safety/HS:SO1 (EL2904)
//     Pumps room star point - coupler (EK1101)/Pumps room star point - Slot 2 (EK1122)/HS: Hydraulics & Safety/HS:SL (EL6900)/ConnectionInputs/Message_91 TxPDO <-> Module 1 (FSOES)/RxPDO/FSOE
//   ECAT (EtherCAT) <-> ECAT (EtherCAT)/Pumps room star point - coupler (EK1101)/Pumps room star point - Slot 2 (EK1122)/PG: Pumps Group/PG:SI1 (EL1904)
//     Pumps room star point - coupler (EK1101)/Pumps room star point - Slot 2 (EK1122)/HS: Hydraulics & Safety/HS:SL (EL6900)/ConnectionInputs/Message_78 TxPDO <-> Module 1 (FSOES)/RxPDO/FSOE
//   ECAT (EtherCAT) <-> ECAT (EtherCAT)/Pumps room star point - coupler (EK1101)/Pumps room star point - Slot 2 (EK1122)/PG: Pumps Group/PG:SI2 (EL1904)
//     Pumps room star point - coupler (EK1101)/Pumps room star point - Slot 2 (EK1122)/HS: Hydraulics & Safety/HS:SL (EL6900)/ConnectionInputs/Message_79 TxPDO <-> Module 1 (FSOES)/RxPDO/FSOE
//   ECAT (EtherCAT) <-> ECAT (EtherCAT)/Pumps room star point - coupler (EK1101)/Pumps room star point - Slot 2 (EK1122)/PG: Pumps Group/PG:SI3 (EL1904)
//     Pumps room star point - coupler (EK1101)/Pumps room star point - Slot 2 (EK1122)/HS: Hydraulics & Safety/HS:SL (EL6900)/ConnectionInputs/Message_80 TxPDO <-> Module 1 (FSOES)/RxPDO/FSOE
//   ECAT (EtherCAT) <-> ECAT (EtherCAT)/Pumps room star point - coupler (EK1101)/Pumps room star point - Slot 3 (EK1122)/DA: Dome Access/DA:SI1 (EL1904)
//     Pumps room star point - coupler (EK1101)/Pumps room star point - Slot 2 (EK1122)/HS: Hydraulics & Safety/HS:SL (EL6900)/ConnectionInputs/Message_84 TxPDO <-> Module 1 (FSOES)/RxPDO/FSOE
//   ECAT (EtherCAT) <-> Slalib/TelescopePointing
//     InfoData/DcToExtTimeOffset <-> Inputs/fromIo/fromEcatMaster/dcToExtTimeOffset
//     InfoData/DcToTcTimeOffset <-> Inputs/fromIo/fromEcatMaster/dcToTcTimeOffset
//     Pumps room star point - coupler (EK1101)/Pumps room star point - Slot 1 (EK1122)/Timing coupler (EK1100)/Timing Slot 2 (PTP EL6688)/External Sync/External device not connected <-> Inputs/fromIo/fromEL6688/notConnected
//     Pumps room star point - coupler (EK1101)/Pumps room star point - Slot 1 (EK1122)/Timing coupler (EK1100)/Timing Slot 2 (PTP EL6688)/External Sync/External time stamp <-> Inputs/fromIo/fromEL6688/externalTimestamp
//     Pumps room star point - coupler (EK1101)/Pumps room star point - Slot 1 (EK1122)/Timing coupler (EK1100)/Timing Slot 2 (PTP EL6688)/External Sync/Internal time stamp <-> Inputs/fromIo/fromEL6688/internalTimestamp
//     Pumps room star point - coupler (EK1101)/Pumps room star point - Slot 1 (EK1122)/Timing coupler (EK1100)/Timing Slot 2 (PTP EL6688)/External Sync/Time stamp update toggle <-> Inputs/fromIo/fromEL6688/updateToggle
//   Fast SAF/Axes/AZI_ABL <-> ECAT (EtherCAT)/Pumps room star point - coupler (EK1101)/Pumps room star point - Slot 1 (EK1122)/REM star point (CU1128)/REM star point C (CU1128-C)/ABLD (AX5206-0000-0203)
//     Drive/Inputs/In/nState1 <-> AT 1/Drive status word @bit 8
//     Drive/Inputs/In/nState2 <-> AT 1/Drive status word
//     Drive/Outputs/Out/nCtrl1 <-> MDT 1/Master control word @bit 8
//     Enc/Inputs/In/nDataIn1 <-> AT 1/Position feedback value 1 (motor feedback)
//   Fast SAF/Axes/AZI_Physical <-> ECAT (EtherCAT)/Pumps room star point - coupler (EK1101)/Pumps room star point - Slot 1 (EK1122)/REM star point (CU1128)/REM star point C (CU1128-C)/AZID (AX5206-0000-0203)
//     Drive/Inputs/In/nDataIn1 <-> AT 1/Following distance
//     Drive/Inputs/In/nDcOutputTime <-> InfoData/DcOutputShift
//     Drive/Inputs/In/nState1 <-> AT 1/Drive status word @bit 8
//     Drive/Inputs/In/nState2 <-> AT 1/Drive status word
//     Drive/Inputs/In/nState4 @bit 1 <-> WcState/InputToggle
//     Drive/Inputs/In/nState4 <-> WcState/WcState
//     Drive/Outputs/Out/nCtrl1 <-> MDT 1/Master control word @bit 8
//     Drive/Outputs/Out/nDataOut1 <-> MDT 1/Position command value
//     Enc/Inputs/In/nDataIn1 <-> AT 1/Position feedback 1 value
//     Enc/Inputs/In/nDcInputTime <-> InfoData/DcInputShift
//     Enc/Inputs/In/nState4 @bit 1 <-> WcState/InputToggle
//     Enc/Inputs/In/nState4 <-> WcState/WcState
//   Fast SAF/Axes/Cover_Bottom_1 <-> ECAT (EtherCAT)/Pumps room star point - coupler (EK1101)/Pumps room star point - Slot 1 (EK1122)/REM star point (CU1128)/Cover coupler (EK1101)/Cover slot 1 (digital out, EL2008)
//     Drive/Outputs/Out/nCtrl3 <-> Channel 5/Bot_1_Drive_nCtrl3.0
//   Fast SAF/Axes/Cover_Bottom_1 <-> ECAT (EtherCAT)/Pumps room star point - coupler (EK1101)/Pumps room star point - Slot 1 (EK1122)/REM star point (CU1128)/Cover coupler (EK1101)/Cover slot 2 (analog out, EL4008)
//     Drive/Outputs/Out/nDataOut2[0] <-> AO Outputs Channel 5/Bot_1_Drive_nDataOut2_0
//   Fast SAF/Axes/Cover_Bottom_1 <-> ECAT (EtherCAT)/Pumps room star point - coupler (EK1101)/Pumps room star point - Slot 1 (EK1122)/REM star point (CU1128)/Cover coupler (EK1101)/Cover slot 6 (enc bot 1-2, EL5002)
//     Enc/Inputs/In/nDataIn1 <-> SSI Inputs Channel 1/Counter value
//     Enc/Inputs/In/nState1 <-> SSI Inputs Channel 1/Status/Data error
//     Enc/Inputs/In/nState1 @bit 1 <-> SSI Inputs Channel 1/Status/Frame error
//     Enc/Inputs/In/nState1 @bit 2 <-> SSI Inputs Channel 1/Status/Power failure
//     Enc/Inputs/In/nState4 @bit 1 <-> WcState/InputToggle
//     Enc/Inputs/In/nState4 <-> WcState/WcState
//   Fast SAF/Axes/Cover_Bottom_2 <-> ECAT (EtherCAT)/Pumps room star point - coupler (EK1101)/Pumps room star point - Slot 1 (EK1122)/REM star point (CU1128)/Cover coupler (EK1101)/Cover slot 1 (digital out, EL2008)
//     Drive/Outputs/Out/nCtrl3 <-> Channel 6/Bot_2_Drive_nCtrl3.0
//   Fast SAF/Axes/Cover_Bottom_2 <-> ECAT (EtherCAT)/Pumps room star point - coupler (EK1101)/Pumps room star point - Slot 1 (EK1122)/REM star point (CU1128)/Cover coupler (EK1101)/Cover slot 2 (analog out, EL4008)
//     Drive/Outputs/Out/nDataOut2[0] <-> AO Outputs Channel 6/Bot_2_Drive_nDataOut2_0
//   Fast SAF/Axes/Cover_Bottom_2 <-> ECAT (EtherCAT)/Pumps room star point - coupler (EK1101)/Pumps room star point - Slot 1 (EK1122)/REM star point (CU1128)/Cover coupler (EK1101)/Cover slot 6 (enc bot 1-2, EL5002)
//     Enc/Inputs/In/nDataIn1 <-> SSI Inputs Channel 2/Counter value
//     Enc/Inputs/In/nState1 <-> SSI Inputs Channel 2/Status/Data error
//     Enc/Inputs/In/nState1 @bit 1 <-> SSI Inputs Channel 2/Status/Frame error
//     Enc/Inputs/In/nState1 @bit 2 <-> SSI Inputs Channel 2/Status/Power failure
//     Enc/Inputs/In/nState4 @bit 1 <-> WcState/InputToggle
//     Enc/Inputs/In/nState4 <-> WcState/WcState
//   Fast SAF/Axes/Cover_Bottom_3 <-> ECAT (EtherCAT)/Pumps room star point - coupler (EK1101)/Pumps room star point - Slot 1 (EK1122)/REM star point (CU1128)/Cover coupler (EK1101)/Cover slot 1 (digital out, EL2008)
//     Drive/Outputs/Out/nCtrl3 <-> Channel 7/Bot_3_Drive_nCtrl3.0
//   Fast SAF/Axes/Cover_Bottom_3 <-> ECAT (EtherCAT)/Pumps room star point - coupler (EK1101)/Pumps room star point - Slot 1 (EK1122)/REM star point (CU1128)/Cover coupler (EK1101)/Cover slot 2 (analog out, EL4008)
//     Drive/Outputs/Out/nDataOut2[0] <-> AO Outputs Channel 7/Bot_3_Drive_nDataOut2_0
//   Fast SAF/Axes/Cover_Bottom_3 <-> ECAT (EtherCAT)/Pumps room star point - coupler (EK1101)/Pumps room star point - Slot 1 (EK1122)/REM star point (CU1128)/Cover coupler (EK1101)/Cover slot 7 (enc bot 3-4, EL5002)
//     Enc/Inputs/In/nDataIn1 <-> SSI Inputs Channel 1/Counter value
//     Enc/Inputs/In/nState1 <-> SSI Inputs Channel 1/Status/Data error
//     Enc/Inputs/In/nState1 @bit 1 <-> SSI Inputs Channel 1/Status/Frame error
//     Enc/Inputs/In/nState1 @bit 2 <-> SSI Inputs Channel 1/Status/Power failure
//     Enc/Inputs/In/nState4 @bit 1 <-> WcState/InputToggle
//     Enc/Inputs/In/nState4 <-> WcState/WcState
//   Fast SAF/Axes/Cover_Bottom_4 <-> ECAT (EtherCAT)/Pumps room star point - coupler (EK1101)/Pumps room star point - Slot 1 (EK1122)/REM star point (CU1128)/Cover coupler (EK1101)/Cover slot 1 (digital out, EL2008)
//     Drive/Outputs/Out/nCtrl3 <-> Channel 8/Bot_4_Drive_nCtrl3.0
//   Fast SAF/Axes/Cover_Bottom_4 <-> ECAT (EtherCAT)/Pumps room star point - coupler (EK1101)/Pumps room star point - Slot 1 (EK1122)/REM star point (CU1128)/Cover coupler (EK1101)/Cover slot 2 (analog out, EL4008)
//     Drive/Outputs/Out/nDataOut2[0] <-> AO Outputs Channel 8/Bot_4_Drive_nDataOut2_0
//   Fast SAF/Axes/Cover_Bottom_4 <-> ECAT (EtherCAT)/Pumps room star point - coupler (EK1101)/Pumps room star point - Slot 1 (EK1122)/REM star point (CU1128)/Cover coupler (EK1101)/Cover slot 7 (enc bot 3-4, EL5002)
//     Enc/Inputs/In/nDataIn1 <-> SSI Inputs Channel 2/Counter value
//     Enc/Inputs/In/nState1 <-> SSI Inputs Channel 2/Status/Data error
//     Enc/Inputs/In/nState1 @bit 1 <-> SSI Inputs Channel 2/Status/Frame error
//     Enc/Inputs/In/nState1 @bit 2 <-> SSI Inputs Channel 2/Status/Power failure
//     Enc/Inputs/In/nState4 @bit 1 <-> WcState/InputToggle
//     Enc/Inputs/In/nState4 <-> WcState/WcState
//   Fast SAF/Axes/Cover_Top_1 <-> ECAT (EtherCAT)/Pumps room star point - coupler (EK1101)/Pumps room star point - Slot 1 (EK1122)/REM star point (CU1128)/Cover coupler (EK1101)/Cover slot 1 (digital out, EL2008)
//     Drive/Outputs/Out/nCtrl3 <-> Channel 1/Top_1_Drive_nCtrl3.0
//   Fast SAF/Axes/Cover_Top_1 <-> ECAT (EtherCAT)/Pumps room star point - coupler (EK1101)/Pumps room star point - Slot 1 (EK1122)/REM star point (CU1128)/Cover coupler (EK1101)/Cover slot 2 (analog out, EL4008)
//     Drive/Outputs/Out/nDataOut2[0] <-> AO Outputs Channel 1/Top_1_Drive_nDataOut2_0
//   Fast SAF/Axes/Cover_Top_1 <-> ECAT (EtherCAT)/Pumps room star point - coupler (EK1101)/Pumps room star point - Slot 1 (EK1122)/REM star point (CU1128)/Cover coupler (EK1101)/Cover slot 4 (enc top 1-2, EL5002)
//     Enc/Inputs/In/nDataIn1 <-> SSI Inputs Channel 1/Counter value
//     Enc/Inputs/In/nState1 <-> SSI Inputs Channel 1/Status/Data error
//     Enc/Inputs/In/nState1 @bit 1 <-> SSI Inputs Channel 1/Status/Frame error
//     Enc/Inputs/In/nState1 @bit 2 <-> SSI Inputs Channel 1/Status/Power failure
//     Enc/Inputs/In/nState4 @bit 1 <-> WcState/InputToggle
//     Enc/Inputs/In/nState4 <-> WcState/WcState
//   Fast SAF/Axes/Cover_Top_2 <-> ECAT (EtherCAT)/Pumps room star point - coupler (EK1101)/Pumps room star point - Slot 1 (EK1122)/REM star point (CU1128)/Cover coupler (EK1101)/Cover slot 1 (digital out, EL2008)
//     Drive/Outputs/Out/nCtrl3 <-> Channel 2/Top_2_Drive_nCtrl3.0
//   Fast SAF/Axes/Cover_Top_2 <-> ECAT (EtherCAT)/Pumps room star point - coupler (EK1101)/Pumps room star point - Slot 1 (EK1122)/REM star point (CU1128)/Cover coupler (EK1101)/Cover slot 2 (analog out, EL4008)
//     Drive/Outputs/Out/nDataOut2[0] <-> AO Outputs Channel 2/Top_2_Drive_nDataOut2_0
//   Fast SAF/Axes/Cover_Top_2 <-> ECAT (EtherCAT)/Pumps room star point - coupler (EK1101)/Pumps room star point - Slot 1 (EK1122)/REM star point (CU1128)/Cover coupler (EK1101)/Cover slot 4 (enc top 1-2, EL5002)
//     Enc/Inputs/In/nDataIn1 <-> SSI Inputs Channel 2/Counter value
//     Enc/Inputs/In/nState1 <-> SSI Inputs Channel 2/Status/Data error
//     Enc/Inputs/In/nState1 @bit 1 <-> SSI Inputs Channel 2/Status/Frame error
//     Enc/Inputs/In/nState1 @bit 2 <-> SSI Inputs Channel 2/Status/Power failure
//     Enc/Inputs/In/nState4 @bit 1 <-> WcState/InputToggle
//     Enc/Inputs/In/nState4 <-> WcState/WcState
//   Fast SAF/Axes/Cover_Top_3 <-> ECAT (EtherCAT)/Pumps room star point - coupler (EK1101)/Pumps room star point - Slot 1 (EK1122)/REM star point (CU1128)/Cover coupler (EK1101)/Cover slot 1 (digital out, EL2008)
//     Drive/Outputs/Out/nCtrl3 <-> Channel 3/Top_3_Drive_nCtrl3.0
//   Fast SAF/Axes/Cover_Top_3 <-> ECAT (EtherCAT)/Pumps room star point - coupler (EK1101)/Pumps room star point - Slot 1 (EK1122)/REM star point (CU1128)/Cover coupler (EK1101)/Cover slot 2 (analog out, EL4008)
//     Drive/Outputs/Out/nDataOut2[0] <-> AO Outputs Channel 3/Top_3_Drive_nDataOut2_0
//   Fast SAF/Axes/Cover_Top_3 <-> ECAT (EtherCAT)/Pumps room star point - coupler (EK1101)/Pumps room star point - Slot 1 (EK1122)/REM star point (CU1128)/Cover coupler (EK1101)/Cover slot 5 (enc top 3-4, EL5002)
//     Enc/Inputs/In/nDataIn1 <-> SSI Inputs Channel 1/Counter value
//     Enc/Inputs/In/nState1 <-> SSI Inputs Channel 1/Status/Data error
//     Enc/Inputs/In/nState1 @bit 1 <-> SSI Inputs Channel 1/Status/Frame error
//     Enc/Inputs/In/nState1 @bit 2 <-> SSI Inputs Channel 1/Status/Power failure
//     Enc/Inputs/In/nState4 @bit 1 <-> WcState/InputToggle
//     Enc/Inputs/In/nState4 <-> WcState/WcState
//   Fast SAF/Axes/Cover_Top_4 <-> ECAT (EtherCAT)/Pumps room star point - coupler (EK1101)/Pumps room star point - Slot 1 (EK1122)/REM star point (CU1128)/Cover coupler (EK1101)/Cover slot 1 (digital out, EL2008)
//     Drive/Outputs/Out/nCtrl3 <-> Channel 4/Top_4_Drive_nCtrl3.0
//   Fast SAF/Axes/Cover_Top_4 <-> ECAT (EtherCAT)/Pumps room star point - coupler (EK1101)/Pumps room star point - Slot 1 (EK1122)/REM star point (CU1128)/Cover coupler (EK1101)/Cover slot 2 (analog out, EL4008)
//     Drive/Outputs/Out/nDataOut2[0] <-> AO Outputs Channel 4/Top_4_Drive_nDataOut2_0
//   Fast SAF/Axes/Cover_Top_4 <-> ECAT (EtherCAT)/Pumps room star point - coupler (EK1101)/Pumps room star point - Slot 1 (EK1122)/REM star point (CU1128)/Cover coupler (EK1101)/Cover slot 5 (enc top 3-4, EL5002)
//     Enc/Inputs/In/nDataIn1 <-> SSI Inputs Channel 2/Counter value
//     Enc/Inputs/In/nState1 <-> SSI Inputs Channel 2/Status/Data error
//     Enc/Inputs/In/nState1 @bit 1 <-> SSI Inputs Channel 2/Status/Frame error
//     Enc/Inputs/In/nState1 @bit 2 <-> SSI Inputs Channel 2/Status/Power failure
//     Enc/Inputs/In/nState4 @bit 1 <-> WcState/InputToggle
//     Enc/Inputs/In/nState4 <-> WcState/WcState
//   Fast SAF/Axes/ELE_Physical <-> ECAT (EtherCAT)/Pumps room star point - coupler (EK1101)/Pumps room star point - Slot 1 (EK1122)/REM star point (CU1128)/REM star point C (CU1128-C)/ELED (AX5206-0000-0203)
//     Drive/Inputs/In/nDataIn1 <-> AT 1/Following distance
//     Drive/Inputs/In/nDcOutputTime <-> InfoData/DcOutputShift
//     Drive/Inputs/In/nState1 <-> AT 1/Drive status word @bit 8
//     Drive/Inputs/In/nState2 <-> AT 1/Drive status word
//     Drive/Inputs/In/nState4 @bit 1 <-> WcState/InputToggle
//     Drive/Inputs/In/nState4 <-> WcState/WcState
//     Drive/Outputs/Out/nCtrl1 <-> MDT 1/Master control word @bit 8
//     Drive/Outputs/Out/nDataOut1 <-> MDT 1/Position command value
//     Enc/Inputs/In/nDataIn1 <-> AT 1/Position feedback 1 value
//     Enc/Inputs/In/nDcInputTime <-> InfoData/DcInputShift
//     Enc/Inputs/In/nState4 @bit 1 <-> WcState/InputToggle
//     Enc/Inputs/In/nState4 <-> WcState/WcState
//   Fast SAF/Axes/M3_RotationAntiBacklash <-> M3 CANopen bus/Box 3 (MCBL3006S-CO) - ROTABL
//     Drive/Inputs/In/nState1 <-> TxPDO 1/Inputs/Statusword
//     Drive/Inputs/In/nState2 <-> TxPDO 1/Inputs/Statusword @bit 8
//     Drive/Outputs/Out/nCtrl1 <-> RxPDO 1/Outputs/Controlword
//     Drive/Outputs/Out/nCtrl2 <-> RxPDO 1/Outputs/Controlword @bit 8
//     Drive/Outputs/Out/nDataOut2 <-> RxPDO 2/Outputs/Target Velocity
//     Enc/Inputs/In/nDataIn1 <-> TxPDO 2/Inputs/Position Actual Value
//   Fast SAF/Axes/M3_RotationPosHall <-> M3 CANopen bus/Box 2 (MCBL3006S-CO) - ROTPOS
//     Enc/Inputs/In/nDataIn1 <-> TxPDO 2/Inputs/Position Actual Value
//   Fast SAF/Axes/M3_RotationPositioning <-> ECAT (EtherCAT)/Pumps room star point - coupler (EK1101)/Pumps room star point - Slot 1 (EK1122)/REM star point (CU1128)/REM star point B (CU1128-B)/M3 coupler (EK1100)/M3 Slot 3 (encoder EL5001)
//     Enc/Inputs/In/nDataIn1 <-> SSI Inputs/Counter value
//     Enc/Inputs/In/nState1 <-> SSI Inputs/Status/Data error
//     Enc/Inputs/In/nState1 @bit 1 <-> SSI Inputs/Status/Frame error
//     Enc/Inputs/In/nState1 @bit 2 <-> SSI Inputs/Status/Power failure
//     Enc/Inputs/In/nState4 @bit 1 <-> WcState/InputToggle
//     Enc/Inputs/In/nState4 <-> WcState/WcState
//   Fast SAF/Axes/M3_RotationPositioning <-> M3 CANopen bus/Box 2 (MCBL3006S-CO) - ROTPOS
//     Drive/Inputs/In/nState1 <-> TxPDO 1/Inputs/Statusword
//     Drive/Inputs/In/nState2 <-> TxPDO 1/Inputs/Statusword @bit 8
//     Drive/Outputs/Out/nCtrl1 <-> RxPDO 1/Outputs/Controlword
//     Drive/Outputs/Out/nCtrl2 <-> RxPDO 1/Outputs/Controlword @bit 8
//     Drive/Outputs/Out/nDataOut2 <-> RxPDO 2/Outputs/Target Velocity
//   Fast SAF/Axes/M3_Translation <-> ECAT (EtherCAT)/Pumps room star point - coupler (EK1101)/Pumps room star point - Slot 1 (EK1122)/REM star point (CU1128)/REM star point B (CU1128-B)/M3 coupler (EK1100)/M3 Slot 2 (encoder EL5101)
//     Enc/Inputs/In/nDataIn1[0] <-> ENC Status compact/Counter value
//     Enc/Inputs/In/nDataIn2[0] <-> ENC Status compact/Latch value
//     Enc/Inputs/In/nState1 @bit 4 <-> ENC Status compact/Status/Counter overflow
//     Enc/Inputs/In/nState1 @bit 3 <-> ENC Status compact/Status/Counter underflow
//     Enc/Inputs/In/nState1 @bit 7 <-> ENC Status compact/Status/Extrapolation stall
//     Enc/Inputs/In/nState1 <-> ENC Status compact/Status/Latch C valid
//     Enc/Inputs/In/nState1 @bit 1 <-> ENC Status compact/Status/Latch extern valid
//     Enc/Inputs/In/nState1 @bit 6 <-> ENC Status compact/Status/Open circuit
//     Enc/Inputs/In/nState1 @bit 2 <-> ENC Status compact/Status/Set counter done
//     Enc/Inputs/In/nState1 @bit 5 <-> ENC Status compact/Status/Status of input status
//     Enc/Inputs/In/nState2 @bit 4 <-> ENC Status compact/Status/Status of extern latch
//     Enc/Inputs/In/nState2 <-> ENC Status compact/Status/Status of input A
//     Enc/Inputs/In/nState2 @bit 1 <-> ENC Status compact/Status/Status of input B
//     Enc/Inputs/In/nState2 @bit 2 <-> ENC Status compact/Status/Status of input C
//     Enc/Inputs/In/nState2 @bit 3 <-> ENC Status compact/Status/Status of input gate
//     Enc/Inputs/In/nState4 @bit 1 <-> WcState/InputToggle
//     Enc/Inputs/In/nState4 <-> WcState/WcState
//     Enc/Outputs/Out/nCtrl1 <-> ENC Control compact/Control/Enable latch C
//     Enc/Outputs/Out/nCtrl1 @bit 3 <-> ENC Control compact/Control/Enable latch extern on negative edge
//     Enc/Outputs/Out/nCtrl1 @bit 1 <-> ENC Control compact/Control/Enable latch extern on positive edge
//     Enc/Outputs/Out/nCtrl1 @bit 2 <-> ENC Control compact/Control/Set counter
//     Enc/Outputs/Out/nDataOut1[0] <-> ENC Control compact/Set counter value
//   Fast SAF/Axes/M3_Translation <-> M3 CANopen bus/Box 1 (MCBL3006S-CO) - LINMOT
//     Drive/Inputs/In/nState1 <-> TxPDO 1/Inputs/Statusword
//     Drive/Inputs/In/nState2 <-> TxPDO 1/Inputs/Statusword @bit 8
//     Drive/Outputs/Out/nCtrl1 <-> RxPDO 1/Outputs/Controlword
//     Drive/Outputs/Out/nCtrl2 <-> RxPDO 1/Outputs/Controlword @bit 8
//     Drive/Outputs/Out/nDataOut2 <-> RxPDO 2/Outputs/Target Velocity
//   Fast SAF/Axes/ROC_Physical <-> ECAT (EtherCAT)/Pumps room star point - coupler (EK1101)/Pumps room star point - Slot 1 (EK1122)/REM star point (CU1128)/REM star point C (CU1128-C)/AZID (AX5206-0000-0203)
//     Drive/Inputs/In/nDataIn1 <-> AT 2/Following distance
//     Drive/Inputs/In/nDcOutputTime <-> InfoData/DcOutputShift
//     Drive/Inputs/In/nState1 <-> AT 2/Drive status word @bit 8
//     Drive/Inputs/In/nState2 <-> AT 2/Drive status word
//     Drive/Inputs/In/nState4 @bit 1 <-> WcState/InputToggle
//     Drive/Inputs/In/nState4 <-> WcState/WcState
//     Drive/Outputs/Out/nCtrl1 <-> MDT 2/Master control word @bit 8
//     Drive/Outputs/Out/nDataOut1 <-> MDT 2/Position command value
//     Enc/Inputs/In/nDataIn1 <-> AT 2/Position feedback 1 value
//     Enc/Inputs/In/nDcInputTime <-> InfoData/DcInputShift
//     Enc/Inputs/In/nState4 @bit 1 <-> WcState/InputToggle
//     Enc/Inputs/In/nState4 <-> WcState/WcState
//   Fast SAF/Axes/RON_Physical <-> ECAT (EtherCAT)/Pumps room star point - coupler (EK1101)/Pumps room star point - Slot 1 (EK1122)/REM star point (CU1128)/REM star point C (CU1128-C)/ABLD (AX5206-0000-0203)
//     Drive/Inputs/In/nDataIn1 <-> AT 2/Following distance
//     Drive/Inputs/In/nDataIn3[0] <-> AT 2/Torque feedback value
//     Drive/Inputs/In/nDcOutputTime <-> InfoData/DcOutputShift
//     Drive/Inputs/In/nState1 <-> AT 2/Drive status word @bit 8
//     Drive/Inputs/In/nState2 <-> AT 2/Drive status word
//     Drive/Inputs/In/nState4 @bit 1 <-> WcState/InputToggle
//     Drive/Inputs/In/nState4 <-> WcState/WcState
//     Drive/Outputs/Out/nCtrl1 <-> MDT 2/Master control word @bit 8
//     Drive/Outputs/Out/nDataOut1 <-> MDT 2/Position command value
//     Enc/Inputs/In/nDataIn1 <-> AT 2/Position feedback value 1 (motor feedback)
//     Enc/Inputs/In/nDcInputTime <-> InfoData/DcInputShift
//     Enc/Inputs/In/nState4 @bit 1 <-> WcState/InputToggle
//     Enc/Inputs/In/nState4 <-> WcState/WcState
//   MTCS/MTCS Instance <-> ECAT (EtherCAT)
//     PlcTask Inputs/GLOBAL.mtcs.parts.services.parts.timing.fromEcatMaster/dcToExtTimeOffset <-> InfoData/DcToExtTimeOffset
//     PlcTask Inputs/GLOBAL.mtcs.parts.services.parts.timing.fromEcatMaster/dcToTcTimeOffset <-> InfoData/DcToTcTimeOffset
//   MTCS/MTCS Instance <-> ECAT (EtherCAT)/Pumps room star point - coupler (EK1101)/Pumps room star point - Slot 1 (EK1122)/REM star point (CU1128)/Cover coupler (EK1101)
//     PlcTask Inputs/GLOBAL.mtcs.parts.cover.parts.io.parts.coupler.infoData <-> InfoData/State
//     PlcTask Inputs/GLOBAL.mtcs.parts.cover.parts.io.parts.coupler.wcState <-> WcState/WcState
//   MTCS/MTCS Instance <-> ECAT (EtherCAT)/Pumps room star point - coupler (EK1101)/Pumps room star point - Slot 1 (EK1122)/REM star point (CU1128)/Cover coupler (EK1101)/Cover slot 1 (digital out, EL2008)
//     PlcTask Inputs/GLOBAL.mtcs.parts.cover.parts.io.parts.slot1.infoData <-> InfoData/State
//     PlcTask Inputs/GLOBAL.mtcs.parts.cover.parts.io.parts.slot1.wcState <-> WcState/WcState
//   MTCS/MTCS Instance <-> ECAT (EtherCAT)/Pumps room star point - coupler (EK1101)/Pumps room star point - Slot 1 (EK1122)/REM star point (CU1128)/Cover coupler (EK1101)/Cover slot 10 (relays bot 1-2, EL2622)
//     PlcTask Inputs/GLOBAL.mtcs.parts.cover.parts.io.parts.slot10.infoData <-> InfoData/State
//     PlcTask Inputs/GLOBAL.mtcs.parts.cover.parts.io.parts.slot10.wcState <-> WcState/WcState
//     PlcTask Outputs/GLOBAL.mtcs.parts.cover.parts.bottom.parts.p1.parts.motorRelay.digitalOutput <-> Channel 1/Output
//     PlcTask Outputs/GLOBAL.mtcs.parts.cover.parts.bottom.parts.p2.parts.motorRelay.digitalOutput <-> Channel 2/Output
//   MTCS/MTCS Instance <-> ECAT (EtherCAT)/Pumps room star point - coupler (EK1101)/Pumps room star point - Slot 1 (EK1122)/REM star point (CU1128)/Cover coupler (EK1101)/Cover slot 11 (relays bot 3-4, EL2622)
//     PlcTask Inputs/GLOBAL.mtcs.parts.cover.parts.io.parts.slot11.infoData <-> InfoData/State
